LIN {X 0,Y 523.904,Z 120.849,A -85,B 0,C 180,E1 -4806.401,E2 -4806.401} C_VEL
LIN {X 0,Y 523.923,Z 120.845,A -85,B 0,C 180,E1 -4809.085,E2 -4809.085} C_VEL
LIN {X 0,Y 523.952,Z 120.843,A -85,B 0,C 180,E1 -4812.119,E2 -4812.119} C_VEL
LIN {X 0,Y 523.947,Z 120.843,A -85,B 0,C 180,E1 -4815.31,E2 -4815.31} C_VEL
LIN {X 0,Y 523.957,Z 120.839,A -85,B 0,C 180,E1 -4818.69,E2 -4818.69} C_VEL
LIN {X 0,Y 523.918,Z 120.847,A -85,B 0,C 180,E1 -4821.081,E2 -4821.081} C_VEL
LIN {X 0,Y 523.902,Z 120.847,A -85,B 0,C 180,E1 -4823.825,E2 -4823.825} C_VEL
LIN {X 0,Y 523.914,Z 120.844,A -85,B 0,C 180,E1 -4826.634,E2 -4826.634} C_VEL
LIN {X 0,Y 523.95,Z 120.845,A -85,B 0,C 180,E1 -4829.355,E2 -4829.355} C_VEL
LIN {X 0,Y 523.96,Z 120.838,A -85,B 0,C 180,E1 -4832.286,E2 -4832.286} C_VEL
LIN {X 0,Y 523.904,Z 120.849,A -85,B 0,C 180,E1 -4835.427,E2 -4835.427} C_VEL
LIN {X 0,Y 523.94,Z 120.841,A -85,B 0,C 180,E1 -4837.94,E2 -4837.94} C_VEL
LIN {X 0,Y 523.971,Z 120.837,A -85,B 0,C 180,E1 -4840.408,E2 -4840.408} C_VEL
LIN {X 0,Y 523.945,Z 120.848,A -85,B 0,C 180,E1 -4842.837,E2 -4842.837} C_VEL
LIN {X 0,Y 523.976,Z 120.84,A -85,B 0,C 180,E1 -4845.236,E2 -4845.236} C_VEL
LIN {X 0,Y 524.016,Z 120.834,A -85,B 0,C 180,E1 -4848.394,E2 -4848.394} C_VEL
LIN {X 0,Y 523.988,Z 120.833,A -85,B 0,C 180,E1 -4851.516,E2 -4851.516} C_VEL
LIN {X 0,Y 524.069,Z 120.832,A -85,B 0,C 180,E1 -4854.614,E2 -4854.614} C_VEL
LIN {X 0,Y 524.111,Z 120.82,A -85,B 0,C 180,E1 -4857.695,E2 -4857.695} C_VEL
LIN {X 0,Y 524.12,Z 120.822,A -85,B 0,C 180,E1 -4860.768,E2 -4860.768} C_VEL
LIN {X 0,Y 524.006,Z 120.833,A -85,B 0,C 180,E1 -4863.075,E2 -4863.075} C_VEL
LIN {X 0,Y 524.067,Z 120.824,A -85,B 0,C 180,E1 -4865.387,E2 -4865.387} C_VEL
LIN {X 0,Y 523.963,Z 120.84,A -85,B 0,C 180,E1 -4868.485,E2 -4868.485} C_VEL
LIN {X 0,Y 524.001,Z 120.838,A -85,B 0,C 180,E1 -4871.736,E2 -4871.736} C_VEL
LIN {X 0,Y 523.99,Z 120.835,A -85,B 0,C 180,E1 -4875.049,E2 -4875.049} C_VEL
LIN {X 0,Y 523.916,Z 120.852,A -85,B 0,C 180,E1 -4877.971,E2 -4877.971} C_VEL
LIN {X 0,Y 523.951,Z 120.84,A -85,B 0,C 180,E1 -4880.411,E2 -4880.411} C_VEL
LIN {X 0,Y 523.909,Z 120.845,A -85,B 0,C 180,E1 -4882.894,E2 -4882.894} C_VEL
LIN {X 0,Y 523.902,Z 120.849,A -85,B 0,C 180,E1 -4885.421,E2 -4885.421} C_VEL
LIN {X 0,Y 523.907,Z 120.848,A -85,B 0,C 180,E1 -4888.003,E2 -4888.003} C_VEL
LIN {X 0,Y 523.91,Z 120.846,A -85,B 0,C 180,E1 -4890.848,E2 -4890.848} C_VEL
LIN {X 0,Y 523.927,Z 120.846,A -85,B 0,C 180,E1 -4893.729,E2 -4893.729} C_VEL
LIN {X 0,Y 523.888,Z 120.847,A -85,B 0,C 180,E1 -4896.399,E2 -4896.399} C_VEL
LIN {X 0,Y 523.91,Z 120.85,A -85,B 0,C 180,E1 -4899.086,E2 -4899.086} C_VEL
LIN {X 0,Y 523.892,Z 120.846,A -85,B 0,C 180,E1 -4902.125,E2 -4902.125} C_VEL
LIN {X 0,Y 523.935,Z 120.848,A -85,B 0,C 180,E1 -4905.311,E2 -4905.311} C_VEL
LIN {X 0,Y 523.878,Z 120.854,A -85,B 0,C 180,E1 -4906.888,E2 -4906.888} C_VEL
LIN {X 0,Y 523.199,Z 120.937,A -85,B 0,C 180,E1 -4907.529,E2 -4907.529} C_VEL
LIN {X 0,Y 520.357,Z 121.291,A -85,B 0,C 180,E1 -4908.571,E2 -4908.571} C_VEL
LIN {X 0,Y 517.966,Z 121.59,A -85,B 0,C 180,E1 -4909.41,E2 -4909.41} C_VEL
LIN {X 0,Y 516.94,Z 121.715,A -85,B 0,C 180,E1 -4910.058,E2 -4910.058} C_VEL
LIN {X 0,Y 516.856,Z 121.726,A -85,B 0,C 180,E1 -4910.277,E2 -4910.277} C_VEL
LIN {X 0,Y 516.815,Z 121.733,A -85,B 0,C 180,E1 -4913.249,E2 -4913.249} C_VEL
LIN {X 0,Y 516.867,Z 121.725,A -85,B 0,C 180,E1 -4916.117,E2 -4916.117} C_VEL
LIN {X 0,Y 516.848,Z 121.726,A -85,B 0,C 180,E1 -4918.944,E2 -4918.944} C_VEL
LIN {X 0,Y 516.855,Z 121.729,A -85,B 0,C 180,E1 -4922.11,E2 -4922.11} C_VEL
LIN {X 0,Y 516.85,Z 121.746,A -85,B 0,C 180,E1 -4924.907,E2 -4924.907} C_VEL
LIN {X 0,Y 519.11,Z 132.074,A -85,B 0,C 180,E1 -4926.671,E2 -4926.671} C_VEL
LIN {X 0,Y 518.957,Z 140.283,A -85,B 0,C 180,E1 -4927.947,E2 -4927.947} C_VEL
LIN {X 0,Y 518.924,Z 142.324,A -85,B 0,C 180,E1 -4928.26,E2 -4928.26} C_VEL
LIN {X 0,Y 522.001,Z 156.207,A -85,B 0,C 180,E1 -4928.604,E2 -4928.604} C_VEL
LIN {X 0,Y 520.908,Z 307.341,A -85,B 0,C 180,E1 -4930.757,E2 -4930.757} C_VEL
LIN {X 0,Y 520.622,Z 323.147,A -85,B 0,C 180,E1 -4931.147,E2 -4931.147} C_VEL
LIN {X 0,Y 520.269,Z 338.38,A -85,B 0,C 180,E1 -4931.695,E2 -4931.695} C_VEL
LIN {X 0,Y 519.864,Z 351.067,A -85,B 0,C 180,E1 -4932.291,E2 -4932.291} C_VEL
LIN {X 0,Y 519.302,Z 364.673,A -85,B 0,C 180,E1 -4933.084,E2 -4933.084} C_VEL
LIN {X 0,Y 518.776,Z 377.627,A -85,B 0,C 180,E1 -4934.012,E2 -4934.012} C_VEL
LIN {X 0,Y 518.258,Z 389.833,A -85,B 0,C 180,E1 -4935.069,E2 -4935.069} C_VEL
LIN {X 0,Y 517.798,Z 401.302,A -85,B 0,C 180,E1 -4936.259,E2 -4936.259} C_VEL
LIN {X 0,Y 517.363,Z 410.954,A -85,B 0,C 180,E1 -4937.447,E2 -4937.447} C_VEL
LIN {X 0,Y 517.036,Z 420.409,A -85,B 0,C 180,E1 -4938.831,E2 -4938.831} C_VEL
LIN {X 0,Y 516.755,Z 428.281,A -85,B 0,C 180,E1 -4940.212,E2 -4940.212} C_VEL
LIN {X 0,Y 516.546,Z 435.629,A -85,B 0,C 180,E1 -4941.787,E2 -4941.787} C_VEL
LIN {X 0,Y 516.391,Z 441.827,A -85,B 0,C 180,E1 -4943.474,E2 -4943.474} C_VEL
LIN {X 0,Y 516.383,Z 444.913,A -85,B 0,C 180,E1 -4944.533,E2 -4944.533} C_VEL
LIN {X 0,Y 516.327,Z 448.416,A -85,B 0,C 180,E1 -4946.098,E2 -4946.098} C_VEL
LIN {X 0,Y 516.259,Z 450.736,A -85,B 0,C 180,E1 -4947.659,E2 -4947.659} C_VEL
LIN {X 0,Y 516.157,Z 451.927,A -85,B 0,C 180,E1 -4949.22,E2 -4949.22} C_VEL
LIN {X 0,Y 516.158,Z 451.946,A -85,B 0,C 180,E1 -4950.78,E2 -4950.78} C_VEL
LIN {X 0,Y 516.259,Z 450.832,A -85,B 0,C 180,E1 -4952.341,E2 -4952.341} C_VEL
LIN {X 0,Y 516.327,Z 448.586,A -85,B 0,C 180,E1 -4953.902,E2 -4953.902} C_VEL
LIN {X 0,Y 516.38,Z 445.154,A -85,B 0,C 180,E1 -4955.467,E2 -4955.467} C_VEL
LIN {X 0,Y 516.407,Z 440.456,A -85,B 0,C 180,E1 -4957.036,E2 -4957.036} C_VEL
LIN {X 0,Y 516.586,Z 434.365,A -85,B 0,C 180,E1 -4958.607,E2 -4958.607} C_VEL
LIN {X 0,Y 516.804,Z 426.696,A -85,B 0,C 180,E1 -4960.183,E2 -4960.183} C_VEL
LIN {X 0,Y 517.084,Z 418.515,A -85,B 0,C 180,E1 -4961.565,E2 -4961.565} C_VEL
LIN {X 0,Y 517.468,Z 408.661,A -85,B 0,C 180,E1 -4962.95,E2 -4962.95} C_VEL
LIN {X 0,Y 517.877,Z 398.555,A -85,B 0,C 180,E1 -4964.139,E2 -4964.139} C_VEL
LIN {X 0,Y 518.392,Z 386.643,A -85,B 0,C 180,E1 -4965.318,E2 -4965.318} C_VEL
LIN {X 0,Y 518.979,Z 373.3,A -85,B 0,C 180,E1 -4966.411,E2 -4966.411} C_VEL
LIN {X 0,Y 519.534,Z 359.772,A -85,B 0,C 180,E1 -4967.314,E2 -4967.314} C_VEL
LIN {X 0,Y 520.028,Z 344.864,A -85,B 0,C 180,E1 -4968.11,E2 -4968.11} C_VEL
LIN {X 0,Y 520.469,Z 329.611,A -85,B 0,C 180,E1 -4968.731,E2 -4968.731} C_VEL
LIN {X 0,Y 520.798,Z 314.908,A -85,B 0,C 180,E1 -4969.167,E2 -4969.167} C_VEL
LIN {X 0,Y 521,Z 299.457,A -85,B 0,C 180,E1 -4969.463,E2 -4969.463} C_VEL
LIN {X 0,Y 522.003,Z 157.022,A -85,B 0,C 180,E1 -4971.475,E2 -4971.475} C_VEL
LIN {X 0,Y 520.545,Z 149.408,A -85,B 0,C 180,E1 -4971.649,E2 -4971.649} C_VEL
LIN {X 0,Y 518.91,Z 142.309,A -85,B 0,C 180,E1 -4971.832,E2 -4971.832} C_VEL
LIN {X 0,Y 519.187,Z 132.644,A -85,B 0,C 180,E1 -4973.325,E2 -4973.325} C_VEL
LIN {X 0,Y 516.847,Z 121.733,A -85,B 0,C 180,E1 -4975.2,E2 -4975.2} C_VEL
LIN {X 0,Y 516.829,Z 121.731,A -85,B 0,C 180,E1 -4978.421,E2 -4978.421} C_VEL
LIN {X 0,Y 516.848,Z 121.732,A -85,B 0,C 180,E1 -4981.112,E2 -4981.112} C_VEL
LIN {X 0,Y 516.869,Z 121.724,A -85,B 0,C 180,E1 -4983.959,E2 -4983.959} C_VEL
LIN {X 0,Y 516.8,Z 121.735,A -85,B 0,C 180,E1 -4986.753,E2 -4986.753} C_VEL
LIN {X 0,Y 516.825,Z 121.728,A -85,B 0,C 180,E1 -4989.727,E2 -4989.727} C_VEL
LIN {X 0,Y 516.841,Z 121.732,A -85,B 0,C 180,E1 -4992.836,E2 -4992.836} C_VEL
LIN {X 0,Y 516.897,Z 121.727,A -85,B 0,C 180,E1 -4995.007,E2 -4995.007} C_VEL
LIN {X 0,Y 516.847,Z 121.723,A -85,B 0,C 180,E1 -4998.407,E2 -4998.407} C_VEL
LIN {X 0,Y 516.87,Z 121.721,A -85,B 0,C 180,E1 -5001.283,E2 -5001.283} C_VEL
LIN {X 0,Y 516.852,Z 121.731,A -85,B 0,C 180,E1 -5004.673,E2 -5004.673} C_VEL
LIN {X 0,Y 516.893,Z 121.716,A -85,B 0,C 180,E1 -5007.458,E2 -5007.458} C_VEL
LIN {X 0,Y 516.828,Z 121.733,A -85,B 0,C 180,E1 -5010.69,E2 -5010.69} C_VEL
LIN {X 0,Y 516.839,Z 121.725,A -85,B 0,C 180,E1 -5013.337,E2 -5013.337} C_VEL
LIN {X 0,Y 516.884,Z 121.723,A -85,B 0,C 180,E1 -5015.927,E2 -5015.927} C_VEL
LIN {X 0,Y 516.868,Z 121.728,A -85,B 0,C 180,E1 -5018.461,E2 -5018.461} C_VEL
LIN {X 0,Y 516.882,Z 121.72,A -85,B 0,C 180,E1 -5020.954,E2 -5020.954} C_VEL
LIN {X 0,Y 516.834,Z 121.727,A -85,B 0,C 180,E1 -5023.407,E2 -5023.407} C_VEL
LIN {X 0,Y 516.884,Z 121.725,A -85,B 0,C 180,E1 -5025.833,E2 -5025.833} C_VEL
LIN {X 0,Y 516.951,Z 121.712,A -85,B 0,C 180,E1 -5029.028,E2 -5029.028} C_VEL
LIN {X 0,Y 516.927,Z 121.719,A -85,B 0,C 180,E1 -5032.186,E2 -5032.186} C_VEL
LIN {X 0,Y 516.989,Z 121.706,A -85,B 0,C 180,E1 -5034.539,E2 -5034.539} C_VEL
LIN {X 0,Y 517.077,Z 121.704,A -85,B 0,C 180,E1 -5037.663,E2 -5037.663} C_VEL
LIN {X 0,Y 517.072,Z 121.698,A -85,B 0,C 180,E1 -5040,E2 -5040} C_VEL
LIN {X 0,Y 517.082,Z 121.696,A -85,B 0,C 180,E1 -5042.337,E2 -5042.337} C_VEL
LIN {X 0,Y 517.015,Z 121.709,A -85,B 0,C 180,E1 -5045.46,E2 -5045.46} C_VEL
LIN {X 0,Y 516.956,Z 121.711,A -85,B 0,C 180,E1 -5048.6,E2 -5048.6} C_VEL
LIN {X 0,Y 516.956,Z 121.714,A -85,B 0,C 180,E1 -5051.807,E2 -5051.807} C_VEL
LIN {X 0,Y 516.94,Z 121.72,A -85,B 0,C 180,E1 -5055.143,E2 -5055.143} C_VEL
LIN {X 0,Y 516.915,Z 121.714,A -85,B 0,C 180,E1 -5058.222,E2 -5058.222} C_VEL
LIN {X 0,Y 516.908,Z 121.722,A -85,B 0,C 180,E1 -5060.702,E2 -5060.702} C_VEL
LIN {X 0,Y 516.886,Z 121.721,A -85,B 0,C 180,E1 -5064.073,E2 -5064.073} C_VEL
LIN {X 0,Y 516.897,Z 121.723,A -85,B 0,C 180,E1 -5066.659,E2 -5066.659} C_VEL
LIN {X 0,Y 516.911,Z 121.718,A -85,B 0,C 180,E1 -5069.523,E2 -5069.523} C_VEL
LIN {X 0,Y 516.896,Z 121.726,A -85,B 0,C 180,E1 -5072.543,E2 -5072.543} C_VEL
LIN {X 0,Y 516.867,Z 121.723,A -85,B 0,C 180,E1 -5075.329,E2 -5075.329} C_VEL
LIN {X 0,Y 516.881,Z 121.721,A -85,B 0,C 180,E1 -5077.943,E2 -5077.943} C_VEL
LIN {X 0,Y 516.884,Z 121.726,A -85,B 0,C 180,E1 -5080.742,E2 -5080.742} C_VEL
LIN {X 0,Y 516.884,Z 121.724,A -85,B 0,C 180,E1 -5082.831,E2 -5082.831} C_VEL
LIN {X 0,Y 516.896,Z 121.72,A -85,B 0,C 180,E1 -5085.007,E2 -5085.007} C_VEL
LIN {X 0,Y 516.914,Z 121.721,A -85,B 0,C 180,E1 -5088.399,E2 -5088.399} C_VEL
LIN {X 0,Y 516.883,Z 121.721,A -85,B 0,C 180,E1 -5091.284,E2 -5091.284} C_VEL
LIN {X 0,Y 516.872,Z 121.729,A -85,B 0,C 180,E1 -5094.219,E2 -5094.219} C_VEL
LIN {X 0,Y 516.896,Z 121.721,A -85,B 0,C 180,E1 -5097.053,E2 -5097.053} C_VEL
LIN {X 0,Y 516.893,Z 121.725,A -85,B 0,C 180,E1 -5099.796,E2 -5099.796} C_VEL
LIN {X 0,Y 516.97,Z 121.904,A -85,B 0,C 180,E1 -5101.763,E2 -5101.763} C_VEL
LIN {X 0,Y 519.924,Z 134.919,A -85,B 0,C 180,E1 -5103.724,E2 -5103.724} C_VEL
LIN {X 0,Y 519.285,Z 155.389,A -85,B 0,C 180,E1 -5106.468,E2 -5106.468} C_VEL
LIN {X 0,Y 518.846,Z 168.536,A -85,B 0,C 180,E1 -5108.206,E2 -5108.206} C_VEL
LIN {X 0,Y 521.856,Z 183.857,A -85,B 0,C 180,E1 -5108.559,E2 -5108.559} C_VEL
LIN {X 0,Y 520.934,Z 318.473,A -85,B 0,C 180,E1 -5110.458,E2 -5110.458} C_VEL
LIN {X 0,Y 520.766,Z 339.002,A -85,B 0,C 180,E1 -5110.799,E2 -5110.799} C_VEL
LIN {X 0,Y 520.416,Z 353.58,A -85,B 0,C 180,E1 -5111.19,E2 -5111.19} C_VEL
LIN {X 0,Y 519.992,Z 368.148,A -85,B 0,C 180,E1 -5111.736,E2 -5111.736} C_VEL
LIN {X 0,Y 519.528,Z 381.49,A -85,B 0,C 180,E1 -5112.381,E2 -5112.381} C_VEL
LIN {X 0,Y 519.024,Z 394.711,A -85,B 0,C 180,E1 -5113.176,E2 -5113.176} C_VEL
LIN {X 0,Y 518.531,Z 407.433,A -85,B 0,C 180,E1 -5114.108,E2 -5114.108} C_VEL
LIN {X 0,Y 517.946,Z 420.434,A -85,B 0,C 180,E1 -5115.261,E2 -5115.261} C_VEL
LIN {X 0,Y 517.52,Z 431.632,A -85,B 0,C 180,E1 -5116.452,E2 -5116.452} C_VEL
LIN {X 0,Y 517.1,Z 442.501,A -85,B 0,C 180,E1 -5117.839,E2 -5117.839} C_VEL
LIN {X 0,Y 516.872,Z 451.552,A -85,B 0,C 180,E1 -5119.224,E2 -5119.224} C_VEL
LIN {X 0,Y 516.575,Z 459.057,A -85,B 0,C 180,E1 -5120.604,E2 -5120.604} C_VEL
LIN {X 0,Y 516.435,Z 466.064,A -85,B 0,C 180,E1 -5122.178,E2 -5122.178} C_VEL
LIN {X 0,Y 516.36,Z 471.573,A -85,B 0,C 180,E1 -5123.749,E2 -5123.749} C_VEL
LIN {X 0,Y 516.239,Z 475.735,A -85,B 0,C 180,E1 -5125.315,E2 -5125.315} C_VEL
LIN {X 0,Y 516.27,Z 478.657,A -85,B 0,C 180,E1 -5126.879,E2 -5126.879} C_VEL
LIN {X 0,Y 516.189,Z 480.396,A -85,B 0,C 180,E1 -5128.44,E2 -5128.44} C_VEL
LIN {X 0,Y 516.152,Z 480.992,A -85,B 0,C 180,E1 -5130,E2 -5130} C_VEL
LIN {X 0,Y 516.189,Z 480.394,A -85,B 0,C 180,E1 -5131.56,E2 -5131.56} C_VEL
LIN {X 0,Y 516.27,Z 478.652,A -85,B 0,C 180,E1 -5133.121,E2 -5133.121} C_VEL
LIN {X 0,Y 516.239,Z 475.733,A -85,B 0,C 180,E1 -5134.685,E2 -5134.685} C_VEL
LIN {X 0,Y 516.365,Z 471.577,A -85,B 0,C 180,E1 -5136.251,E2 -5136.251} C_VEL
LIN {X 0,Y 516.435,Z 466.065,A -85,B 0,C 180,E1 -5137.821,E2 -5137.821} C_VEL
LIN {X 0,Y 516.575,Z 459.051,A -85,B 0,C 180,E1 -5139.396,E2 -5139.396} C_VEL
LIN {X 0,Y 516.858,Z 451.548,A -85,B 0,C 180,E1 -5140.776,E2 -5140.776} C_VEL
LIN {X 0,Y 517.089,Z 442.772,A -85,B 0,C 180,E1 -5142.122,E2 -5142.122} C_VEL
LIN {X 0,Y 517.473,Z 433.272,A -85,B 0,C 180,E1 -5143.349,E2 -5143.349} C_VEL
LIN {X 0,Y 517.871,Z 422.4,A -85,B 0,C 180,E1 -5144.54,E2 -5144.54} C_VEL
LIN {X 0,Y 518.336,Z 411.334,A -85,B 0,C 180,E1 -5145.565,E2 -5145.565} C_VEL
LIN {X 0,Y 518.829,Z 399.006,A -85,B 0,C 180,E1 -5146.527,E2 -5146.527} C_VEL
LIN {X 0,Y 519.381,Z 386.798,A -85,B 0,C 180,E1 -5147.319,E2 -5147.319} C_VEL
LIN {X 0,Y 519.837,Z 372.671,A -85,B 0,C 180,E1 -5148.066,E2 -5148.066} C_VEL
LIN {X 0,Y 520.323,Z 358.14,A -85,B 0,C 180,E1 -5148.66,E2 -5148.66} C_VEL
LIN {X 0,Y 520.674,Z 342.45,A -85,B 0,C 180,E1 -5149.127,E2 -5149.127} C_VEL
LIN {X 0,Y 520.934,Z 326.359,A -85,B 0,C 180,E1 -5149.429,E2 -5149.429} C_VEL
LIN {X 0,Y 521.902,Z 184.332,A -85,B 0,C 180,E1 -5151.432,E2 -5151.432} C_VEL
LIN {X 0,Y 518.854,Z 168.468,A -85,B 0,C 180,E1 -5151.798,E2 -5151.798} C_VEL
LIN {X 0,Y 519.503,Z 149.094,A -85,B 0,C 180,E1 -5154.369,E2 -5154.369} C_VEL
LIN {X 0,Y 519.914,Z 134.915,A -85,B 0,C 180,E1 -5156.276,E2 -5156.276} C_VEL
LIN {X 0,Y 516.925,Z 121.723,A -85,B 0,C 180,E1 -5158.275,E2 -5158.275} C_VEL
LIN {X 0,Y 516.89,Z 121.721,A -85,B 0,C 180,E1 -5161.11,E2 -5161.11} C_VEL
LIN {X 0,Y 516.908,Z 121.723,A -85,B 0,C 180,E1 -5163.966,E2 -5163.966} C_VEL
LIN {X 0,Y 516.877,Z 121.722,A -85,B 0,C 180,E1 -5166.746,E2 -5166.746} C_VEL
LIN {X 0,Y 516.883,Z 121.727,A -85,B 0,C 180,E1 -5169.721,E2 -5169.721} C_VEL
LIN {X 0,Y 516.912,Z 121.725,A -85,B 0,C 180,E1 -5171.775,E2 -5171.775} C_VEL
LIN {X 0,Y 516.896,Z 121.719,A -85,B 0,C 180,E1 -5175.007,E2 -5175.007} C_VEL
LIN {X 0,Y 516.914,Z 121.716,A -85,B 0,C 180,E1 -5178.399,E2 -5178.399} C_VEL
LIN {X 0,Y 516.881,Z 121.726,A -85,B 0,C 180,E1 -5181.284,E2 -5181.284} C_VEL
LIN {X 0,Y 516.872,Z 121.72,A -85,B 0,C 180,E1 -5184.22,E2 -5184.22} C_VEL
LIN {X 0,Y 516.882,Z 121.724,A -85,B 0,C 180,E1 -5187.052,E2 -5187.052} C_VEL
LIN {X 0,Y 516.888,Z 121.72,A -85,B 0,C 180,E1 -5189.796,E2 -5189.796} C_VEL
LIN {X 0,Y 516.912,Z 121.717,A -85,B 0,C 180,E1 -5192.467,E2 -5192.467} C_VEL
LIN {X 0,Y 516.874,Z 121.722,A -85,B 0,C 180,E1 -5195.645,E2 -5195.645} C_VEL
LIN {X 0,Y 516.887,Z 121.722,A -85,B 0,C 180,E1 -5198.462,E2 -5198.462} C_VEL
LIN {X 0,Y 516.894,Z 121.726,A -85,B 0,C 180,E1 -5200.955,E2 -5200.955} C_VEL
LIN {X 0,Y 516.899,Z 121.718,A -85,B 0,C 180,E1 -5203.41,E2 -5203.41} C_VEL
LIN {X 0,Y 516.885,Z 121.72,A -85,B 0,C 180,E1 -5205.833,E2 -5205.833} C_VEL
LIN {X 0,Y 516.952,Z 121.716,A -85,B 0,C 180,E1 -5209.028,E2 -5209.028} C_VEL
LIN {X 0,Y 516.946,Z 121.713,A -85,B 0,C 180,E1 -5212.186,E2 -5212.186} C_VEL
LIN {X 0,Y 517.015,Z 121.711,A -85,B 0,C 180,E1 -5214.54,E2 -5214.54} C_VEL
LIN {X 0,Y 517.082,Z 121.696,A -85,B 0,C 180,E1 -5217.663,E2 -5217.663} C_VEL
LIN {X 0,Y 517.091,Z 121.697,A -85,B 0,C 180,E1 -5220.779,E2 -5220.779} C_VEL
LIN {X 0,Y 516.95,Z 121.712,A -85,B 0,C 180,E1 -5223.117,E2 -5223.117} C_VEL
LIN {X 0,Y 516.974,Z 121.717,A -85,B 0,C 180,E1 -5226.244,E2 -5226.244} C_VEL
LIN {X 0,Y 516.939,Z 121.711,A -85,B 0,C 180,E1 -5229.39,E2 -5229.39} C_VEL
LIN {X 0,Y 516.955,Z 121.717,A -85,B 0,C 180,E1 -5231.807,E2 -5231.807} C_VEL
LIN {X 0,Y 516.942,Z 121.713,A -85,B 0,C 180,E1 -5235.144,E2 -5235.144} C_VEL
LIN {X 0,Y 516.878,Z 121.725,A -85,B 0,C 180,E1 -5238.224,E2 -5238.224} C_VEL
LIN {X 0,Y 516.9,Z 121.717,A -85,B 0,C 180,E1 -5240.702,E2 -5240.702} C_VEL
LIN {X 0,Y 516.858,Z 121.726,A -85,B 0,C 180,E1 -5243.224,E2 -5243.224} C_VEL
LIN {X 0,Y 516.883,Z 121.714,A -85,B 0,C 180,E1 -5246.182,E2 -5246.182} C_VEL
LIN {X 0,Y 516.905,Z 121.722,A -85,B 0,C 180,E1 -5249.306,E2 -5249.306} C_VEL
LIN {X 0,Y 516.893,Z 121.719,A -85,B 0,C 180,E1 -5252.542,E2 -5252.542} C_VEL
LIN {X 0,Y 516.856,Z 121.73,A -85,B 0,C 180,E1 -5255.328,E2 -5255.328} C_VEL
LIN {X 0,Y 516.877,Z 121.722,A -85,B 0,C 180,E1 -5257.942,E2 -5257.942} C_VEL
LIN {X 0,Y 516.848,Z 121.726,A -85,B 0,C 180,E1 -5260.745,E2 -5260.745} C_VEL
LIN {X 0,Y 516.881,Z 121.721,A -85,B 0,C 180,E1 -5263.903,E2 -5263.903} C_VEL
LIN {X 0,Y 516.835,Z 121.73,A -85,B 0,C 180,E1 -5266.888,E2 -5266.888} C_VEL
LIN {X 0,Y 516.859,Z 121.726,A -85,B 0,C 180,E1 -5269.593,E2 -5269.593} C_VEL
LIN {X 0,Y 516.856,Z 121.726,A -85,B 0,C 180,E1 -5270.277,E2 -5270.277} C_VEL
LIN {X 0,Y 516.186,Z 121.812,A -85,B 0,C 180,E1 -5270.927,E2 -5270.927} C_VEL
LIN {X 0,Y 513.32,Z 122.169,A -85,B 0,C 180,E1 -5271.982,E2 -5271.982} C_VEL
LIN {X 0,Y 510.897,Z 122.474,A -85,B 0,C 180,E1 -5272.832,E2 -5272.832} C_VEL
LIN {X 0,Y 509.855,Z 122.598,A -85,B 0,C 180,E1 -5273.489,E2 -5273.489} C_VEL
LIN {X 0,Y 509.769,Z 122.607,A -85,B 0,C 180,E1 -5273.711,E2 -5273.711} C_VEL
LIN {X 0,Y 509.824,Z 122.606,A -85,B 0,C 180,E1 -5276.536,E2 -5276.536} C_VEL
LIN {X 0,Y 509.801,Z 122.599,A -85,B 0,C 180,E1 -5279.331,E2 -5279.331} C_VEL
LIN {X 0,Y 509.822,Z 122.605,A -85,B 0,C 180,E1 -5282.05,E2 -5282.05} C_VEL
LIN {X 0,Y 509.826,Z 122.769,A -85,B 0,C 180,E1 -5284.674,E2 -5284.674} C_VEL
LIN {X 0,Y 512.223,Z 133.604,A -85,B 0,C 180,E1 -5286.553,E2 -5286.553} C_VEL
LIN {X 0,Y 512.211,Z 138.98,A -85,B 0,C 180,E1 -5287.407,E2 -5287.407} C_VEL
LIN {X 0,Y 512.063,Z 142.508,A -85,B 0,C 180,E1 -5287.951,E2 -5287.951} C_VEL
LIN {X 0,Y 515.364,Z 156.872,A -85,B 0,C 180,E1 -5288.32,E2 -5288.32} C_VEL
LIN {X 0,Y 514.4,Z 284.989,A -85,B 0,C 180,E1 -5290.154,E2 -5290.154} C_VEL
LIN {X 0,Y 514.17,Z 309.47,A -85,B 0,C 180,E1 -5290.538,E2 -5290.538} C_VEL
LIN {X 0,Y 513.881,Z 324.887,A -85,B 0,C 180,E1 -5290.942,E2 -5290.942} C_VEL
LIN {X 0,Y 513.499,Z 339.718,A -85,B 0,C 180,E1 -5291.497,E2 -5291.497} C_VEL
LIN {X 0,Y 513.045,Z 353.179,A -85,B 0,C 180,E1 -5292.151,E2 -5292.151} C_VEL
LIN {X 0,Y 512.46,Z 366.447,A -85,B 0,C 180,E1 -5292.954,E2 -5292.954} C_VEL
LIN {X 0,Y 511.837,Z 380.179,A -85,B 0,C 180,E1 -5293.98,E2 -5293.98} C_VEL
LIN {X 0,Y 511.288,Z 392.149,A -85,B 0,C 180,E1 -5295.064,E2 -5295.064} C_VEL
LIN {X 0,Y 510.805,Z 403.276,A -85,B 0,C 180,E1 -5296.271,E2 -5296.271} C_VEL
LIN {X 0,Y 510.278,Z 414.357,A -85,B 0,C 180,E1 -5297.714,E2 -5297.714} C_VEL
LIN {X 0,Y 509.98,Z 423.052,A -85,B 0,C 180,E1 -5299.077,E2 -5299.077} C_VEL
LIN {X 0,Y 509.678,Z 430.483,A -85,B 0,C 180,E1 -5300.475,E2 -5300.475} C_VEL
LIN {X 0,Y 509.453,Z 437.431,A -85,B 0,C 180,E1 -5302.071,E2 -5302.071} C_VEL
LIN {X 0,Y 509.315,Z 442.893,A -85,B 0,C 180,E1 -5303.662,E2 -5303.662} C_VEL
LIN {X 0,Y 509.166,Z 447.02,A -85,B 0,C 180,E1 -5305.249,E2 -5305.249} C_VEL
LIN {X 0,Y 509.189,Z 449.92,A -85,B 0,C 180,E1 -5306.835,E2 -5306.835} C_VEL
LIN {X 0,Y 509.11,Z 451.67,A -85,B 0,C 180,E1 -5308.418,E2 -5308.418} C_VEL
LIN {X 0,Y 509.066,Z 452.284,A -85,B 0,C 180,E1 -5310,E2 -5310} C_VEL
LIN {X 0,Y 509.111,Z 451.727,A -85,B 0,C 180,E1 -5311.582,E2 -5311.582} C_VEL
LIN {X 0,Y 509.19,Z 450.051,A -85,B 0,C 180,E1 -5313.165,E2 -5313.165} C_VEL
LIN {X 0,Y 509.165,Z 447.223,A -85,B 0,C 180,E1 -5314.751,E2 -5314.751} C_VEL
LIN {X 0,Y 509.307,Z 443.168,A -85,B 0,C 180,E1 -5316.338,E2 -5316.338} C_VEL
LIN {X 0,Y 509.453,Z 437.791,A -85,B 0,C 180,E1 -5317.929,E2 -5317.929} C_VEL
LIN {X 0,Y 509.666,Z 430.939,A -85,B 0,C 180,E1 -5319.525,E2 -5319.525} C_VEL
LIN {X 0,Y 509.965,Z 422.384,A -85,B 0,C 180,E1 -5321.124,E2 -5321.124} C_VEL
LIN {X 0,Y 510.326,Z 413.291,A -85,B 0,C 180,E1 -5322.527,E2 -5322.527} C_VEL
LIN {X 0,Y 510.749,Z 404.014,A -85,B 0,C 180,E1 -5323.731,E2 -5323.731} C_VEL
LIN {X 0,Y 511.279,Z 392.026,A -85,B 0,C 180,E1 -5325.038,E2 -5325.038} C_VEL
LIN {X 0,Y 511.915,Z 379.005,A -85,B 0,C 180,E1 -5326.204,E2 -5326.204} C_VEL
LIN {X 0,Y 512.476,Z 366.26,A -85,B 0,C 180,E1 -5327.148,E2 -5327.148} C_VEL
LIN {X 0,Y 513.014,Z 352.963,A -85,B 0,C 180,E1 -5327.953,E2 -5327.953} C_VEL
LIN {X 0,Y 513.555,Z 338.286,A -85,B 0,C 180,E1 -5328.656,E2 -5328.656} C_VEL
LIN {X 0,Y 513.941,Z 323.44,A -85,B 0,C 180,E1 -5329.194,E2 -5329.194} C_VEL
LIN {X 0,Y 514.232,Z 307.532,A -85,B 0,C 180,E1 -5329.593,E2 -5329.593} C_VEL
LIN {X 0,Y 515.379,Z 157.183,A -85,B 0,C 180,E1 -5331.765,E2 -5331.765} C_VEL
LIN {X 0,Y 512.066,Z 142.467,A -85,B 0,C 180,E1 -5332.144,E2 -5332.144} C_VEL
LIN {X 0,Y 512.317,Z 134.163,A -85,B 0,C 180,E1 -5333.442,E2 -5333.442} C_VEL
LIN {X 0,Y 509.801,Z 122.612,A -85,B 0,C 180,E1 -5335.464,E2 -5335.464} C_VEL
LIN {X 0,Y 509.808,Z 122.607,A -85,B 0,C 180,E1 -5338.082,E2 -5338.082} C_VEL
LIN {X 0,Y 509.815,Z 122.609,A -85,B 0,C 180,E1 -5341.274,E2 -5341.274} C_VEL
LIN {X 0,Y 509.821,Z 122.602,A -85,B 0,C 180,E1 -5344.416,E2 -5344.416} C_VEL
LIN {X 0,Y 509.763,Z 122.616,A -85,B 0,C 180,E1 -5347.346,E2 -5347.346} C_VEL
LIN {X 0,Y 509.787,Z 122.604,A -85,B 0,C 180,E1 -5350.387,E2 -5350.387} C_VEL
LIN {X 0,Y 509.793,Z 122.606,A -85,B 0,C 180,E1 -5353.575,E2 -5353.575} C_VEL
LIN {X 0,Y 509.792,Z 122.607,A -85,B 0,C 180,E1 -5356.425,E2 -5356.425} C_VEL
LIN {X 0,Y 509.813,Z 122.602,A -85,B 0,C 180,E1 -5359.615,E2 -5359.615} C_VEL
LIN {X 0,Y 509.784,Z 122.605,A -85,B 0,C 180,E1 -5362.656,E2 -5362.656} C_VEL
LIN {X 0,Y 509.84,Z 122.598,A -85,B 0,C 180,E1 -5365.801,E2 -5365.801} C_VEL
LIN {X 0,Y 509.818,Z 122.598,A -85,B 0,C 180,E1 -5368.726,E2 -5368.726} C_VEL
LIN {X 0,Y 509.824,Z 122.603,A -85,B 0,C 180,E1 -5372.05,E2 -5372.05} C_VEL
LIN {X 0,Y 509.803,Z 122.607,A -85,B 0,C 180,E1 -5374.7,E2 -5374.7} C_VEL
LIN {X 0,Y 509.826,Z 122.598,A -85,B 0,C 180,E1 -5377.459,E2 -5377.459} C_VEL
LIN {X 0,Y 509.892,Z 122.595,A -85,B 0,C 180,E1 -5379.844,E2 -5379.844} C_VEL
LIN {X 0,Y 509.849,Z 122.602,A -85,B 0,C 180,E1 -5382.346,E2 -5382.346} C_VEL
LIN {X 0,Y 509.893,Z 122.591,A -85,B 0,C 180,E1 -5384.818,E2 -5384.818} C_VEL
LIN {X 0,Y 509.905,Z 122.597,A -85,B 0,C 180,E1 -5388.124,E2 -5388.124} C_VEL
LIN {X 0,Y 509.887,Z 122.59,A -85,B 0,C 180,E1 -5391.279,E2 -5391.279} C_VEL
LIN {X 0,Y 509.944,Z 122.584,A -85,B 0,C 180,E1 -5394.464,E2 -5394.464} C_VEL
LIN {X 0,Y 510.046,Z 122.579,A -85,B 0,C 180,E1 -5397.631,E2 -5397.631} C_VEL
LIN {X 0,Y 510.041,Z 122.574,A -85,B 0,C 180,E1 -5400,E2 -5400} C_VEL
LIN {X 0,Y 510.052,Z 122.572,A -85,B 0,C 180,E1 -5402.369,E2 -5402.369} C_VEL
LIN {X 0,Y 509.966,Z 122.588,A -85,B 0,C 180,E1 -5405.536,E2 -5405.536} C_VEL
LIN {X 0,Y 509.905,Z 122.59,A -85,B 0,C 180,E1 -5408.72,E2 -5408.72} C_VEL
LIN {X 0,Y 509.907,Z 122.591,A -85,B 0,C 180,E1 -5411.931,E2 -5411.931} C_VEL
LIN {X 0,Y 509.898,Z 122.599,A -85,B 0,C 180,E1 -5415.242,E2 -5415.242} C_VEL
LIN {X 0,Y 509.86,Z 122.594,A -85,B 0,C 180,E1 -5418.484,E2 -5418.484} C_VEL
LIN {X 0,Y 509.849,Z 122.605,A -85,B 0,C 180,E1 -5421.002,E2 -5421.002} C_VEL
LIN {X 0,Y 509.82,Z 122.602,A -85,B 0,C 180,E1 -5423.564,E2 -5423.564} C_VEL
LIN {X 0,Y 509.876,Z 122.594,A -85,B 0,C 180,E1 -5426.369,E2 -5426.369} C_VEL
LIN {X 0,Y 509.854,Z 122.604,A -85,B 0,C 180,E1 -5428.846,E2 -5428.846} C_VEL
LIN {X 0,Y 509.821,Z 122.601,A -85,B 0,C 180,E1 -5431.59,E2 -5431.59} C_VEL
LIN {X 0,Y 509.84,Z 122.6,A -85,B 0,C 180,E1 -5434.414,E2 -5434.414} C_VEL
LIN {X 0,Y 509.818,Z 122.6,A -85,B 0,C 180,E1 -5437.341,E2 -5437.341} C_VEL
LIN {X 0,Y 509.84,Z 122.603,A -85,B 0,C 180,E1 -5440.382,E2 -5440.382} C_VEL
LIN {X 0,Y 509.824,Z 122.601,A -85,B 0,C 180,E1 -5443.062,E2 -5443.062} C_VEL
LIN {X 0,Y 509.824,Z 122.602,A -85,B 0,C 180,E1 -5445.793,E2 -5445.793} C_VEL
LIN {X 0,Y 509.856,Z 122.597,A -85,B 0,C 180,E1 -5448.574,E2 -5448.574} C_VEL
LIN {X 0,Y 509.852,Z 122.6,A -85,B 0,C 180,E1 -5451.786,E2 -5451.786} C_VEL
LIN {X 0,Y 509.831,Z 122.602,A -85,B 0,C 180,E1 -5454.622,E2 -5454.622} C_VEL
LIN {X 0,Y 509.862,Z 122.599,A -85,B 0,C 180,E1 -5457.481,E2 -5457.481} C_VEL
LIN {X 0,Y 509.86,Z 122.602,A -85,B 0,C 180,E1 -5460.274,E2 -5460.274} C_VEL
LIN {X 0,Y 509.89,Z 122.695,A -85,B 0,C 180,E1 -5461.474,E2 -5461.474} C_VEL
LIN {X 0,Y 513.048,Z 136.31,A -85,B 0,C 180,E1 -5463.564,E2 -5463.564} C_VEL
LIN {X 0,Y 512.528,Z 153.629,A -85,B 0,C 180,E1 -5465.924,E2 -5465.924} C_VEL
LIN {X 0,Y 512.008,Z 168.292,A -85,B 0,C 180,E1 -5467.897,E2 -5467.897} C_VEL
LIN {X 0,Y 515.283,Z 185.415,A -85,B 0,C 180,E1 -5468.297,E2 -5468.297} C_VEL
LIN {X 0,Y 514.141,Z 334.566,A -85,B 0,C 180,E1 -5470.446,E2 -5470.446} C_VEL
LIN {X 0,Y 513.801,Z 350.317,A -85,B 0,C 180,E1 -5470.835,E2 -5470.835} C_VEL
LIN {X 0,Y 513.386,Z 364.448,A -85,B 0,C 180,E1 -5471.337,E2 -5471.337} C_VEL
LIN {X 0,Y 512.782,Z 379.472,A -85,B 0,C 180,E1 -5472.038,E2 -5472.038} C_VEL
LIN {X 0,Y 512.234,Z 392.989,A -85,B 0,C 180,E1 -5472.843,E2 -5472.843} C_VEL
LIN {X 0,Y 511.707,Z 405.456,A -85,B 0,C 180,E1 -5473.749,E2 -5473.749} C_VEL
LIN {X 0,Y 511.153,Z 418.137,A -85,B 0,C 180,E1 -5474.856,E2 -5474.856} C_VEL
LIN {X 0,Y 510.615,Z 429.658,A -85,B 0,C 180,E1 -5476.062,E2 -5476.062} C_VEL
LIN {X 0,Y 510.205,Z 439.359,A -85,B 0,C 180,E1 -5477.268,E2 -5477.268} C_VEL
LIN {X 0,Y 509.83,Z 449.043,A -85,B 0,C 180,E1 -5478.697,E2 -5478.697} C_VEL
LIN {X 0,Y 509.562,Z 456.826,A -85,B 0,C 180,E1 -5480.072,E2 -5480.072} C_VEL
LIN {X 0,Y 509.394,Z 464.24,A -85,B 0,C 180,E1 -5481.67,E2 -5481.67} C_VEL
LIN {X 0,Y 509.289,Z 470.122,A -85,B 0,C 180,E1 -5483.264,E2 -5483.264} C_VEL
LIN {X 0,Y 509.263,Z 473.617,A -85,B 0,C 180,E1 -5484.456,E2 -5484.456} C_VEL
LIN {X 0,Y 509.172,Z 477.148,A -85,B 0,C 180,E1 -5486.043,E2 -5486.043} C_VEL
LIN {X 0,Y 509.186,Z 479.473,A -85,B 0,C 180,E1 -5487.627,E2 -5487.627} C_VEL
LIN {X 0,Y 509.07,Z 480.64,A -85,B 0,C 180,E1 -5489.209,E2 -5489.209} C_VEL
LIN {X 0,Y 509.07,Z 480.639,A -85,B 0,C 180,E1 -5490.791,E2 -5490.791} C_VEL
LIN {X 0,Y 509.186,Z 479.469,A -85,B 0,C 180,E1 -5492.373,E2 -5492.373} C_VEL
LIN {X 0,Y 509.172,Z 477.144,A -85,B 0,C 180,E1 -5493.957,E2 -5493.957} C_VEL
LIN {X 0,Y 509.264,Z 473.618,A -85,B 0,C 180,E1 -5495.544,E2 -5495.544} C_VEL
LIN {X 0,Y 509.315,Z 468.799,A -85,B 0,C 180,E1 -5497.134,E2 -5497.134} C_VEL
LIN {X 0,Y 509.453,Z 462.557,A -85,B 0,C 180,E1 -5498.728,E2 -5498.728} C_VEL
LIN {X 0,Y 509.701,Z 454.72,A -85,B 0,C 180,E1 -5500.326,E2 -5500.326} C_VEL
LIN {X 0,Y 509.937,Z 446.321,A -85,B 0,C 180,E1 -5501.738,E2 -5501.738} C_VEL
LIN {X 0,Y 510.339,Z 436.344,A -85,B 0,C 180,E1 -5503.134,E2 -5503.134} C_VEL
LIN {X 0,Y 510.755,Z 426.075,A -85,B 0,C 180,E1 -5504.34,E2 -5504.34} C_VEL
LIN {X 0,Y 511.33,Z 413.429,A -85,B 0,C 180,E1 -5505.585,E2 -5505.585} C_VEL
LIN {X 0,Y 511.917,Z 400.238,A -85,B 0,C 180,E1 -5506.654,E2 -5506.654} C_VEL
LIN {X 0,Y 512.577,Z 386.598,A -85,B 0,C 180,E1 -5507.556,E2 -5507.556} C_VEL
LIN {X 0,Y 513.067,Z 372.471,A -85,B 0,C 180,E1 -5508.312,E2 -5508.312} C_VEL
LIN {X 0,Y 513.586,Z 357.969,A -85,B 0,C 180,E1 -5508.913,E2 -5508.913} C_VEL
LIN {X 0,Y 513.951,Z 342.522,A -85,B 0,C 180,E1 -5509.381,E2 -5509.381} C_VEL
LIN {X 0,Y 514.239,Z 326.159,A -85,B 0,C 180,E1 -5509.693,E2 -5509.693} C_VEL
LIN {X 0,Y 515.303,Z 185.412,A -85,B 0,C 180,E1 -5511.702,E2 -5511.702} C_VEL
LIN {X 0,Y 511.998,Z 168.264,A -85,B 0,C 180,E1 -5512.106,E2 -5512.106} C_VEL
LIN {X 0,Y 512.71,Z 148.903,A -85,B 0,C 180,E1 -5514.714,E2 -5514.714} C_VEL
LIN {X 0,Y 513.037,Z 136.304,A -85,B 0,C 180,E1 -5516.437,E2 -5516.437} C_VEL
LIN {X 0,Y 509.895,Z 122.599,A -85,B 0,C 180,E1 -5518.55,E2 -5518.55} C_VEL
LIN {X 0,Y 509.821,Z 122.603,A -85,B 0,C 180,E1 -5521.59,E2 -5521.59} C_VEL
LIN {X 0,Y 509.848,Z 122.6,A -85,B 0,C 180,E1 -5524.414,E2 -5524.414} C_VEL
LIN {X 0,Y 509.818,Z 122.603,A -85,B 0,C 180,E1 -5527.341,E2 -5527.341} C_VEL
LIN {X 0,Y 509.839,Z 122.6,A -85,B 0,C 180,E1 -5530.382,E2 -5530.382} C_VEL
LIN {X 0,Y 509.825,Z 122.6,A -85,B 0,C 180,E1 -5533.062,E2 -5533.062} C_VEL
LIN {X 0,Y 509.824,Z 122.606,A -85,B 0,C 180,E1 -5535.793,E2 -5535.793} C_VEL
LIN {X 0,Y 509.856,Z 122.595,A -85,B 0,C 180,E1 -5538.575,E2 -5538.575} C_VEL
LIN {X 0,Y 509.852,Z 122.6,A -85,B 0,C 180,E1 -5541.787,E2 -5541.787} C_VEL
LIN {X 0,Y 509.83,Z 122.597,A -85,B 0,C 180,E1 -5544.622,E2 -5544.622} C_VEL
LIN {X 0,Y 509.861,Z 122.601,A -85,B 0,C 180,E1 -5547.481,E2 -5547.481} C_VEL
LIN {X 0,Y 509.86,Z 122.593,A -85,B 0,C 180,E1 -5550.274,E2 -5550.274} C_VEL
LIN {X 0,Y 509.868,Z 122.599,A -85,B 0,C 180,E1 -5552.943,E2 -5552.943} C_VEL
LIN {X 0,Y 509.82,Z 122.6,A -85,B 0,C 180,E1 -5556.436,E2 -5556.436} C_VEL
LIN {X 0,Y 509.917,Z 122.586,A -85,B 0,C 180,E1 -5559.845,E2 -5559.845} C_VEL
LIN {X 0,Y 509.866,Z 122.597,A -85,B 0,C 180,E1 -5563.174,E2 -5563.174} C_VEL
LIN {X 0,Y 509.857,Z 122.596,A -85,B 0,C 180,E1 -5565.634,E2 -5565.634} C_VEL
LIN {X 0,Y 509.915,Z 122.595,A -85,B 0,C 180,E1 -5568.875,E2 -5568.875} C_VEL
LIN {X 0,Y 509.911,Z 122.588,A -85,B 0,C 180,E1 -5572.078,E2 -5572.078} C_VEL
LIN {X 0,Y 509.966,Z 122.59,A -85,B 0,C 180,E1 -5574.464,E2 -5574.464} C_VEL
LIN {X 0,Y 510.052,Z 122.571,A -85,B 0,C 180,E1 -5577.631,E2 -5577.631} C_VEL
LIN {X 0,Y 510.041,Z 122.575,A -85,B 0,C 180,E1 -5580.79,E2 -5580.79} C_VEL
LIN {X 0,Y 510.047,Z 122.58,A -85,B 0,C 180,E1 -5582.369,E2 -5582.369} C_VEL
LIN {X 0,Y 509.964,Z 122.581,A -85,B 0,C 180,E1 -5585.536,E2 -5585.536} C_VEL
LIN {X 0,Y 509.891,Z 122.59,A -85,B 0,C 180,E1 -5588.721,E2 -5588.721} C_VEL
LIN {X 0,Y 509.907,Z 122.596,A -85,B 0,C 180,E1 -5591.932,E2 -5591.932} C_VEL
LIN {X 0,Y 509.898,Z 122.591,A -85,B 0,C 180,E1 -5595.242,E2 -5595.242} C_VEL
LIN {X 0,Y 509.836,Z 122.6,A -85,B 0,C 180,E1 -5598.485,E2 -5598.485} C_VEL
LIN {X 0,Y 509.843,Z 122.596,A -85,B 0,C 180,E1 -5601.002,E2 -5601.002} C_VEL
LIN {X 0,Y 509.82,Z 122.607,A -85,B 0,C 180,E1 -5603.564,E2 -5603.564} C_VEL
LIN {X 0,Y 509.819,Z 122.592,A -85,B 0,C 180,E1 -5606.357,E2 -5606.357} C_VEL
LIN {X 0,Y 509.838,Z 122.598,A -85,B 0,C 180,E1 -5608.847,E2 -5608.847} C_VEL
LIN {X 0,Y 509.814,Z 122.607,A -85,B 0,C 180,E1 -5611.591,E2 -5611.591} C_VEL
LIN {X 0,Y 509.835,Z 122.596,A -85,B 0,C 180,E1 -5614.415,E2 -5614.415} C_VEL
LIN {X 0,Y 509.807,Z 122.608,A -85,B 0,C 180,E1 -5617.342,E2 -5617.342} C_VEL
LIN {X 0,Y 509.813,Z 122.6,A -85,B 0,C 180,E1 -5620.385,E2 -5620.385} C_VEL
LIN {X 0,Y 509.806,Z 122.605,A -85,B 0,C 180,E1 -5623.573,E2 -5623.573} C_VEL
LIN {X 0,Y 509.806,Z 122.603,A -85,B 0,C 180,E1 -5626.426,E2 -5626.426} C_VEL
LIN {X 0,Y 509.813,Z 122.604,A -85,B 0,C 180,E1 -5629.615,E2 -5629.615} C_VEL
LIN {X 0,Y 509.783,Z 122.61,A -85,B 0,C 180,E1 -5632.656,E2 -5632.656} C_VEL
LIN {X 0,Y 509.769,Z 122.607,A -85,B 0,C 180,E1 -5633.711,E2 -5633.711} C_VEL
LIN {X 0,Y 509.109,Z 122.692,A -85,B 0,C 180,E1 -5634.371,E2 -5634.371} C_VEL
LIN {X 0,Y 506.284,Z 123.045,A -85,B 0,C 180,E1 -5635.444,E2 -5635.444} C_VEL
LIN {X 0,Y 503.888,Z 123.345,A -85,B 0,C 180,E1 -5636.307,E2 -5636.307} C_VEL
LIN {X 0,Y 502.847,Z 123.473,A -85,B 0,C 180,E1 -5636.974,E2 -5636.974} C_VEL
LIN {X 0,Y 502.756,Z 123.483,A -85,B 0,C 180,E1 -5637.2,E2 -5637.2} C_VEL
LIN {X 0,Y 502.744,Z 123.476,A -85,B 0,C 180,E1 -5640.079,E2 -5640.079} C_VEL
LIN {X 0,Y 502.768,Z 123.485,A -85,B 0,C 180,E1 -5642.529,E2 -5642.529} C_VEL
LIN {X 0,Y 502.783,Z 123.616,A -85,B 0,C 180,E1 -5644.404,E2 -5644.404} C_VEL
LIN {X 0,Y 505.474,Z 136.043,A -85,B 0,C 180,E1 -5646.585,E2 -5646.585} C_VEL
LIN {X 0,Y 505.253,Z 142.701,A -85,B 0,C 180,E1 -5647.638,E2 -5647.638} C_VEL
LIN {X 0,Y 508.834,Z 158.982,A -85,B 0,C 180,E1 -5648.056,E2 -5648.056} C_VEL
LIN {X 0,Y 507.56,Z 308.005,A -85,B 0,C 180,E1 -5650.235,E2 -5650.235} C_VEL
LIN {X 0,Y 507.218,Z 323.58,A -85,B 0,C 180,E1 -5650.629,E2 -5650.629} C_VEL
LIN {X 0,Y 506.82,Z 338.804,A -85,B 0,C 180,E1 -5651.192,E2 -5651.192} C_VEL
LIN {X 0,Y 506.353,Z 351.488,A -85,B 0,C 180,E1 -5651.803,E2 -5651.803} C_VEL
LIN {X 0,Y 505.72,Z 365.091,A -85,B 0,C 180,E1 -5652.615,E2 -5652.615} C_VEL
LIN {X 0,Y 505.142,Z 377.723,A -85,B 0,C 180,E1 -5653.543,E2 -5653.543} C_VEL
LIN {X 0,Y 504.484,Z 390.246,A -85,B 0,C 180,E1 -5654.651,E2 -5654.651} C_VEL
LIN {X 0,Y 503.934,Z 401.713,A -85,B 0,C 180,E1 -5655.874,E2 -5655.874} C_VEL
LIN {X 0,Y 503.464,Z 411.362,A -85,B 0,C 180,E1 -5657.094,E2 -5657.094} C_VEL
LIN {X 0,Y 503.039,Z 420.969,A -85,B 0,C 180,E1 -5658.542,E2 -5658.542} C_VEL
LIN {X 0,Y 502.66,Z 429.687,A -85,B 0,C 180,E1 -5660.138,E2 -5660.138} C_VEL
LIN {X 0,Y 502.461,Z 436.033,A -85,B 0,C 180,E1 -5661.555,E2 -5661.555} C_VEL
LIN {X 0,Y 502.26,Z 441.987,A -85,B 0,C 180,E1 -5663.21,E2 -5663.21} C_VEL
LIN {X 0,Y 502.262,Z 445.313,A -85,B 0,C 180,E1 -5664.379,E2 -5664.379} C_VEL
LIN {X 0,Y 502.163,Z 448.815,A -85,B 0,C 180,E1 -5665.987,E2 -5665.987} C_VEL
LIN {X 0,Y 502.118,Z 451.134,A -85,B 0,C 180,E1 -5667.593,E2 -5667.593} C_VEL
LIN {X 0,Y 501.988,Z 452.324,A -85,B 0,C 180,E1 -5669.198,E2 -5669.198} C_VEL
LIN {X 0,Y 501.988,Z 452.343,A -85,B 0,C 180,E1 -5670.802,E2 -5670.802} C_VEL
LIN {X 0,Y 502.118,Z 451.227,A -85,B 0,C 180,E1 -5672.407,E2 -5672.407} C_VEL
LIN {X 0,Y 502.163,Z 448.981,A -85,B 0,C 180,E1 -5674.013,E2 -5674.013} C_VEL
LIN {X 0,Y 502.257,Z 445.548,A -85,B 0,C 180,E1 -5675.621,E2 -5675.621} C_VEL
LIN {X 0,Y 502.305,Z 440.85,A -85,B 0,C 180,E1 -5677.234,E2 -5677.234} C_VEL
LIN {X 0,Y 502.486,Z 434.759,A -85,B 0,C 180,E1 -5678.85,E2 -5678.85} C_VEL
LIN {X 0,Y 502.771,Z 427.088,A -85,B 0,C 180,E1 -5680.47,E2 -5680.47} C_VEL
LIN {X 0,Y 503.073,Z 418.802,A -85,B 0,C 180,E1 -5681.909,E2 -5681.909} C_VEL
LIN {X 0,Y 503.568,Z 409.051,A -85,B 0,C 180,E1 -5683.314,E2 -5683.314} C_VEL
LIN {X 0,Y 504.08,Z 398.943,A -85,B 0,C 180,E1 -5684.534,E2 -5684.534} C_VEL
LIN {X 0,Y 504.634,Z 387.6,A -85,B 0,C 180,E1 -5685.691,E2 -5685.691} C_VEL
LIN {X 0,Y 505.246,Z 375.098,A -85,B 0,C 180,E1 -5686.755,E2 -5686.755} C_VEL
LIN {X 0,Y 505.905,Z 361.727,A -85,B 0,C 180,E1 -5687.691,E2 -5687.691} C_VEL
LIN {X 0,Y 506.397,Z 349.239,A -85,B 0,C 180,E1 -5688.405,E2 -5688.405} C_VEL
LIN {X 0,Y 506.963,Z 334.625,A -85,B 0,C 180,E1 -5689.065,E2 -5689.065} C_VEL
LIN {X 0,Y 507.324,Z 319.67,A -85,B 0,C 180,E1 -5689.571,E2 -5689.571} C_VEL
LIN {X 0,Y 507.616,Z 304.447,A -85,B 0,C 180,E1 -5689.917,E2 -5689.917} C_VEL
LIN {X 0,Y 508.844,Z 159.119,A -85,B 0,C 180,E1 -5692.032,E2 -5692.032} C_VEL
LIN {X 0,Y 505.279,Z 142.664,A -85,B 0,C 180,E1 -5692.456,E2 -5692.456} C_VEL
LIN {X 0,Y 505.472,Z 135.939,A -85,B 0,C 180,E1 -5693.523,E2 -5693.523} C_VEL
LIN {X 0,Y 502.785,Z 123.485,A -85,B 0,C 180,E1 -5695.734,E2 -5695.734} C_VEL
LIN {X 0,Y 502.76,Z 123.484,A -85,B 0,C 180,E1 -5698.378,E2 -5698.378} C_VEL
LIN {X 0,Y 502.765,Z 123.488,A -85,B 0,C 180,E1 -5701.493,E2 -5701.493} C_VEL
LIN {X 0,Y 502.773,Z 123.48,A -85,B 0,C 180,E1 -5704.439,E2 -5704.439} C_VEL
LIN {X 0,Y 502.72,Z 123.491,A -85,B 0,C 180,E1 -5707.169,E2 -5707.169} C_VEL
LIN {X 0,Y 502.731,Z 123.482,A -85,B 0,C 180,E1 -5710.021,E2 -5710.021} C_VEL
LIN {X 0,Y 502.74,Z 123.488,A -85,B 0,C 180,E1 -5713.235,E2 -5713.235} C_VEL
LIN {X 0,Y 502.768,Z 123.48,A -85,B 0,C 180,E1 -5715.659,E2 -5715.659} C_VEL
LIN {X 0,Y 502.763,Z 123.486,A -85,B 0,C 180,E1 -5719.013,E2 -5719.013} C_VEL
LIN {X 0,Y 502.761,Z 123.477,A -85,B 0,C 180,E1 -5722.043,E2 -5722.043} C_VEL
LIN {X 0,Y 502.784,Z 123.481,A -85,B 0,C 180,E1 -5725.033,E2 -5725.033} C_VEL
LIN {X 0,Y 502.774,Z 123.475,A -85,B 0,C 180,E1 -5727.915,E2 -5727.915} C_VEL
LIN {X 0,Y 502.754,Z 123.486,A -85,B 0,C 180,E1 -5730.708,E2 -5730.708} C_VEL
LIN {X 0,Y 502.776,Z 123.477,A -85,B 0,C 180,E1 -5733.46,E2 -5733.46} C_VEL
LIN {X 0,Y 502.763,Z 123.484,A -85,B 0,C 180,E1 -5736.085,E2 -5736.085} C_VEL
LIN {X 0,Y 502.833,Z 123.471,A -85,B 0,C 180,E1 -5739.464,E2 -5739.464} C_VEL
LIN {X 0,Y 502.801,Z 123.479,A -85,B 0,C 180,E1 -5742.091,E2 -5742.091} C_VEL
LIN {X 0,Y 502.836,Z 123.471,A -85,B 0,C 180,E1 -5745.429,E2 -5745.429} C_VEL
LIN {X 0,Y 502.879,Z 123.466,A -85,B 0,C 180,E1 -5748.717,E2 -5748.717} C_VEL
LIN {X 0,Y 502.852,Z 123.475,A -85,B 0,C 180,E1 -5751.966,E2 -5751.966} C_VEL
LIN {X 0,Y 502.9,Z 123.462,A -85,B 0,C 180,E1 -5754.386,E2 -5754.386} C_VEL
LIN {X 0,Y 503.013,Z 123.455,A -85,B 0,C 180,E1 -5757.598,E2 -5757.598} C_VEL
LIN {X 0,Y 503.01,Z 123.45,A -85,B 0,C 180,E1 -5760,E2 -5760} C_VEL
LIN {X 0,Y 503.02,Z 123.448,A -85,B 0,C 180,E1 -5762.402,E2 -5762.402} C_VEL
LIN {X 0,Y 502.919,Z 123.466,A -85,B 0,C 180,E1 -5765.614,E2 -5765.614} C_VEL
LIN {X 0,Y 502.865,Z 123.468,A -85,B 0,C 180,E1 -5768.843,E2 -5768.843} C_VEL
LIN {X 0,Y 502.848,Z 123.47,A -85,B 0,C 180,E1 -5772.102,E2 -5772.102} C_VEL
LIN {X 0,Y 502.851,Z 123.475,A -85,B 0,C 180,E1 -5775.4,E2 -5775.4} C_VEL
LIN {X 0,Y 502.825,Z 123.473,A -85,B 0,C 180,E1 -5778.752,E2 -5778.752} C_VEL
LIN {X 0,Y 502.784,Z 123.48,A -85,B 0,C 180,E1 -5781.311,E2 -5781.311} C_VEL
LIN {X 0,Y 502.768,Z 123.48,A -85,B 0,C 180,E1 -5783.915,E2 -5783.915} C_VEL
LIN {X 0,Y 502.837,Z 123.473,A -85,B 0,C 180,E1 -5786.568,E2 -5786.568} C_VEL
LIN {X 0,Y 502.816,Z 123.473,A -85,B 0,C 180,E1 -5789.935,E2 -5789.935} C_VEL
LIN {X 0,Y 502.831,Z 123.472,A -85,B 0,C 180,E1 -5793.031,E2 -5793.031} C_VEL
LIN {X 0,Y 502.775,Z 123.479,A -85,B 0,C 180,E1 -5795.951,E2 -5795.951} C_VEL
LIN {X 0,Y 502.802,Z 123.476,A -85,B 0,C 180,E1 -5798.976,E2 -5798.976} C_VEL
LIN {X 0,Y 502.797,Z 123.48,A -85,B 0,C 180,E1 -5802.139,E2 -5802.139} C_VEL
LIN {X 0,Y 502.787,Z 123.477,A -85,B 0,C 180,E1 -5805.47,E2 -5805.47} C_VEL
LIN {X 0,Y 502.821,Z 123.47,A -85,B 0,C 180,E1 -5808.934,E2 -5808.934} C_VEL
LIN {X 0,Y 502.794,Z 123.481,A -85,B 0,C 180,E1 -5812.046,E2 -5812.046} C_VEL
LIN {X 0,Y 502.8,Z 123.476,A -85,B 0,C 180,E1 -5815.034,E2 -5815.034} C_VEL
LIN {X 0,Y 502.784,Z 123.484,A -85,B 0,C 180,E1 -5817.915,E2 -5817.915} C_VEL
LIN {X 0,Y 502.873,Z 123.546,A -85,B 0,C 180,E1 -5821.189,E2 -5821.189} C_VEL
LIN {X 0,Y 506.214,Z 137.972,A -85,B 0,C 180,E1 -5823.439,E2 -5823.439} C_VEL
LIN {X 0,Y 505.737,Z 153.44,A -85,B 0,C 180,E1 -5825.58,E2 -5825.58} C_VEL
LIN {X 0,Y 505.167,Z 168.045,A -85,B 0,C 180,E1 -5827.575,E2 -5827.575} C_VEL
LIN {X 0,Y 508.703,Z 186.772,A -85,B 0,C 180,E1 -5828.025,E2 -5828.025} C_VEL
LIN {X 0,Y 507.434,Z 334.371,A -85,B 0,C 180,E1 -5830.177,E2 -5830.177} C_VEL
LIN {X 0,Y 507.065,Z 350.12,A -85,B 0,C 180,E1 -5830.571,E2 -5830.571} C_VEL
LIN {X 0,Y 506.618,Z 364.724,A -85,B 0,C 180,E1 -5831.098,E2 -5831.098} C_VEL
LIN {X 0,Y 505.999,Z 379.273,A -85,B 0,C 180,E1 -5831.789,E2 -5831.789} C_VEL
LIN {X 0,Y 505.402,Z 392.789,A -85,B 0,C 180,E1 -5832.604,E2 -5832.604} C_VEL
LIN {X 0,Y 504.819,Z 405.255,A -85,B 0,C 180,E1 -5833.521,E2 -5833.521} C_VEL
LIN {X 0,Y 504.242,Z 417.936,A -85,B 0,C 180,E1 -5834.644,E2 -5834.644} C_VEL
LIN {X 0,Y 503.634,Z 429.457,A -85,B 0,C 180,E1 -5835.865,E2 -5835.865} C_VEL
LIN {X 0,Y 503.192,Z 439.157,A -85,B 0,C 180,E1 -5837.087,E2 -5837.087} C_VEL
LIN {X 0,Y 502.799,Z 448.853,A -85,B 0,C 180,E1 -5838.538,E2 -5838.538} C_VEL
LIN {X 0,Y 502.523,Z 456.626,A -85,B 0,C 180,E1 -5839.932,E2 -5839.932} C_VEL
LIN {X 0,Y 502.323,Z 464.04,A -85,B 0,C 180,E1 -5841.552,E2 -5841.552} C_VEL
LIN {X 0,Y 502.222,Z 469.923,A -85,B 0,C 180,E1 -5843.169,E2 -5843.169} C_VEL
LIN {X 0,Y 502.175,Z 473.418,A -85,B 0,C 180,E1 -5844.378,E2 -5844.378} C_VEL
LIN {X 0,Y 502.069,Z 476.949,A -85,B 0,C 180,E1 -5845.987,E2 -5845.987} C_VEL
LIN {X 0,Y 502.088,Z 479.274,A -85,B 0,C 180,E1 -5847.593,E2 -5847.593} C_VEL
LIN {X 0,Y 501.987,Z 480.441,A -85,B 0,C 180,E1 -5849.198,E2 -5849.198} C_VEL
LIN {X 0,Y 501.987,Z 480.44,A -85,B 0,C 180,E1 -5850.802,E2 -5850.802} C_VEL
LIN {X 0,Y 502.088,Z 479.27,A -85,B 0,C 180,E1 -5852.407,E2 -5852.407} C_VEL
LIN {X 0,Y 502.069,Z 476.944,A -85,B 0,C 180,E1 -5854.013,E2 -5854.013} C_VEL
LIN {X 0,Y 502.176,Z 473.419,A -85,B 0,C 180,E1 -5855.622,E2 -5855.622} C_VEL
LIN {X 0,Y 502.238,Z 468.599,A -85,B 0,C 180,E1 -5857.235,E2 -5857.235} C_VEL
LIN {X 0,Y 502.363,Z 462.356,A -85,B 0,C 180,E1 -5858.852,E2 -5858.852} C_VEL
LIN {X 0,Y 502.634,Z 454.519,A -85,B 0,C 180,E1 -5860.473,E2 -5860.473} C_VEL
LIN {X 0,Y 502.901,Z 445.661,A -85,B 0,C 180,E1 -5861.974,E2 -5861.974} C_VEL
LIN {X 0,Y 503.359,Z 436.143,A -85,B 0,C 180,E1 -5863.319,E2 -5863.319} C_VEL
LIN {X 0,Y 503.805,Z 425.874,A -85,B 0,C 180,E1 -5864.542,E2 -5864.542} C_VEL
LIN {X 0,Y 504.4,Z 413.813,A -85,B 0,C 180,E1 -5865.75,E2 -5865.75} C_VEL
LIN {X 0,Y 504.992,Z 401.373,A -85,B 0,C 180,E1 -5866.785,E2 -5866.785} C_VEL
LIN {X 0,Y 505.68,Z 388.025,A -85,B 0,C 180,E1 -5867.699,E2 -5867.699} C_VEL
LIN {X 0,Y 506.161,Z 375.284,A -85,B 0,C 180,E1 -5868.414,E2 -5868.414} C_VEL
LIN {X 0,Y 506.735,Z 360.948,A -85,B 0,C 180,E1 -5869.05,E2 -5869.05} C_VEL
LIN {X 0,Y 507.141,Z 345.858,A -85,B 0,C 180,E1 -5869.55,E2 -5869.55} C_VEL
LIN {X 0,Y 507.466,Z 331.083,A -85,B 0,C 180,E1 -5869.879,E2 -5869.879} C_VEL
LIN {X 0,Y 508.692,Z 186.574,A -85,B 0,C 180,E1 -5871.978,E2 -5871.978} C_VEL
LIN {X 0,Y 505.146,Z 168.067,A -85,B 0,C 180,E1 -5872.421,E2 -5872.421} C_VEL
LIN {X 0,Y 506.086,Z 145.569,A -85,B 0,C 180,E1 -5875.499,E2 -5875.499} C_VEL
LIN {X 0,Y 506.212,Z 137.964,A -85,B 0,C 180,E1 -5876.561,E2 -5876.561} C_VEL
LIN {X 0,Y 502.837,Z 123.476,A -85,B 0,C 180,E1 -5878.829,E2 -5878.829} C_VEL
LIN {X 0,Y 502.784,Z 123.48,A -85,B 0,C 180,E1 -5882.085,E2 -5882.085} C_VEL
LIN {X 0,Y 502.8,Z 123.475,A -85,B 0,C 180,E1 -5884.966,E2 -5884.966} C_VEL
LIN {X 0,Y 502.794,Z 123.483,A -85,B 0,C 180,E1 -5887.954,E2 -5887.954} C_VEL
LIN {X 0,Y 502.82,Z 123.473,A -85,B 0,C 180,E1 -5891.066,E2 -5891.066} C_VEL
LIN {X 0,Y 502.787,Z 123.476,A -85,B 0,C 180,E1 -5894.53,E2 -5894.53} C_VEL
LIN {X 0,Y 502.796,Z 123.48,A -85,B 0,C 180,E1 -5897.861,E2 -5897.861} C_VEL
LIN {X 0,Y 502.802,Z 123.477,A -85,B 0,C 180,E1 -5901.024,E2 -5901.024} C_VEL
LIN {X 0,Y 502.776,Z 123.476,A -85,B 0,C 180,E1 -5904.169,E2 -5904.169} C_VEL
LIN {X 0,Y 502.832,Z 123.473,A -85,B 0,C 180,E1 -5906.994,E2 -5906.994} C_VEL
LIN {X 0,Y 502.816,Z 123.471,A -85,B 0,C 180,E1 -5910.065,E2 -5910.065} C_VEL
LIN {X 0,Y 502.819,Z 123.473,A -85,B 0,C 180,E1 -5912.532,E2 -5912.532} C_VEL
LIN {X 0,Y 502.772,Z 123.482,A -85,B 0,C 180,E1 -5915.313,E2 -5915.313} C_VEL
LIN {X 0,Y 502.781,Z 123.478,A -85,B 0,C 180,E1 -5917.827,E2 -5917.827} C_VEL
LIN {X 0,Y 502.821,Z 123.471,A -85,B 0,C 180,E1 -5920.4,E2 -5920.4} C_VEL
LIN {X 0,Y 502.813,Z 123.478,A -85,B 0,C 180,E1 -5922.931,E2 -5922.931} C_VEL
LIN {X 0,Y 502.841,Z 123.471,A -85,B 0,C 180,E1 -5925.429,E2 -5925.429} C_VEL
LIN {X 0,Y 502.879,Z 123.471,A -85,B 0,C 180,E1 -5928.717,E2 -5928.717} C_VEL
LIN {X 0,Y 502.874,Z 123.463,A -85,B 0,C 180,E1 -5931.966,E2 -5931.966} C_VEL
LIN {X 0,Y 502.92,Z 123.466,A -85,B 0,C 180,E1 -5934.386,E2 -5934.386} C_VEL
LIN {X 0,Y 503.021,Z 123.447,A -85,B 0,C 180,E1 -5937.598,E2 -5937.598} C_VEL
LIN {X 0,Y 502.992,Z 123.453,A -85,B 0,C 180,E1 -5940.801,E2 -5940.801} C_VEL
LIN {X 0,Y 503.014,Z 123.455,A -85,B 0,C 180,E1 -5942.402,E2 -5942.402} C_VEL
LIN {X 0,Y 502.917,Z 123.46,A -85,B 0,C 180,E1 -5945.614,E2 -5945.614} C_VEL
LIN {X 0,Y 502.854,Z 123.466,A -85,B 0,C 180,E1 -5948.844,E2 -5948.844} C_VEL
LIN {X 0,Y 502.847,Z 123.474,A -85,B 0,C 180,E1 -5952.102,E2 -5952.102} C_VEL
LIN {X 0,Y 502.848,Z 123.471,A -85,B 0,C 180,E1 -5955.4,E2 -5955.4} C_VEL
LIN {X 0,Y 502.809,Z 123.474,A -85,B 0,C 180,E1 -5958.753,E2 -5958.753} C_VEL
LIN {X 0,Y 502.78,Z 123.478,A -85,B 0,C 180,E1 -5961.311,E2 -5961.311} C_VEL
LIN {X 0,Y 502.768,Z 123.482,A -85,B 0,C 180,E1 -5963.915,E2 -5963.915} C_VEL
LIN {X 0,Y 502.785,Z 123.467,A -85,B 0,C 180,E1 -5966.571,E2 -5966.571} C_VEL
LIN {X 0,Y 502.811,Z 123.477,A -85,B 0,C 180,E1 -5969.934,E2 -5969.934} C_VEL
LIN {X 0,Y 502.804,Z 123.477,A -85,B 0,C 180,E1 -5973.033,E2 -5973.033} C_VEL
LIN {X 0,Y 502.764,Z 123.48,A -85,B 0,C 180,E1 -5975.952,E2 -5975.952} C_VEL
LIN {X 0,Y 502.785,Z 123.48,A -85,B 0,C 180,E1 -5978.978,E2 -5978.978} C_VEL
LIN {X 0,Y 502.745,Z 123.48,A -85,B 0,C 180,E1 -5982.192,E2 -5982.192} C_VEL
LIN {X 0,Y 502.787,Z 123.48,A -85,B 0,C 180,E1 -5985.47,E2 -5985.47} C_VEL
LIN {X 0,Y 502.762,Z 123.486,A -85,B 0,C 180,E1 -5988.928,E2 -5988.928} C_VEL
LIN {X 0,Y 502.76,Z 123.48,A -85,B 0,C 180,E1 -5992.043,E2 -5992.043} C_VEL
LIN {X 0,Y 502.78,Z 123.484,A -85,B 0,C 180,E1 -5995.033,E2 -5995.033} C_VEL
LIN {X 0,Y 502.756,Z 123.483,A -85,B 0,C 180,E1 -5997.2,E2 -5997.2} C_VEL
LIN {X 0,Y 502.068,Z 123.569,A -85,B 0,C 180,E1 -5997.869,E2 -5997.869} C_VEL
LIN {X 0,Y 499.197,Z 123.923,A -85,B 0,C 180,E1 -5998.955,E2 -5998.955} C_VEL
LIN {X 0,Y 496.787,Z 124.219,A -85,B 0,C 180,E1 -5999.829,E2 -5999.829} C_VEL
LIN {X 0,Y 495.759,Z 124.347,A -85,B 0,C 180,E1 -6000.505,E2 -6000.505} C_VEL
LIN {X 0,Y 495.679,Z 124.359,A -85,B 0,C 180,E1 -6000.734,E2 -6000.734} C_VEL
LIN {X 0,Y 495.721,Z 124.362,A -85,B 0,C 180,E1 -6003.275,E2 -6003.275} C_VEL
LIN {X 0,Y 495.754,Z 124.476,A -85,B 0,C 180,E1 -6004.128,E2 -6004.128} C_VEL
LIN {X 0,Y 498.574,Z 137.112,A -85,B 0,C 180,E1 -6006.385,E2 -6006.385} C_VEL
LIN {X 0,Y 498.454,Z 142.902,A -85,B 0,C 180,E1 -6007.316,E2 -6007.316} C_VEL
LIN {X 0,Y 502.207,Z 159.15,A -85,B 0,C 180,E1 -6007.75,E2 -6007.75} C_VEL
LIN {X 0,Y 500.991,Z 299.363,A -85,B 0,C 180,E1 -6009.808,E2 -6009.808} C_VEL
LIN {X 0,Y 500.782,Z 315.413,A -85,B 0,C 180,E1 -6010.125,E2 -6010.125} C_VEL
LIN {X 0,Y 500.396,Z 329.877,A -85,B 0,C 180,E1 -6010.568,E2 -6010.568} C_VEL
LIN {X 0,Y 499.856,Z 344.638,A -85,B 0,C 180,E1 -6011.186,E2 -6011.186} C_VEL
LIN {X 0,Y 499.276,Z 358.874,A -85,B 0,C 180,E1 -6011.96,E2 -6011.96} C_VEL
LIN {X 0,Y 498.587,Z 372.557,A -85,B 0,C 180,E1 -6012.887,E2 -6012.887} C_VEL
LIN {X 0,Y 497.902,Z 385.602,A -85,B 0,C 180,E1 -6013.971,E2 -6013.971} C_VEL
LIN {X 0,Y 497.331,Z 396.444,A -85,B 0,C 180,E1 -6015.055,E2 -6015.055} C_VEL
LIN {X 0,Y 496.769,Z 406.94,A -85,B 0,C 180,E1 -6016.292,E2 -6016.292} C_VEL
LIN {X 0,Y 496.19,Z 417.185,A -85,B 0,C 180,E1 -6017.733,E2 -6017.733} C_VEL
LIN {X 0,Y 495.86,Z 425.687,A -85,B 0,C 180,E1 -6019.176,E2 -6019.176} C_VEL
LIN {X 0,Y 495.534,Z 432.764,A -85,B 0,C 180,E1 -6020.613,E2 -6020.613} C_VEL
LIN {X 0,Y 495.306,Z 439.328,A -85,B 0,C 180,E1 -6022.253,E2 -6022.253} C_VEL
LIN {X 0,Y 495.18,Z 444.058,A -85,B 0,C 180,E1 -6023.736,E2 -6023.736} C_VEL
LIN {X 0,Y 495.019,Z 447.42,A -85,B 0,C 180,E1 -6025.113,E2 -6025.113} C_VEL
LIN {X 0,Y 495.035,Z 450.318,A -85,B 0,C 180,E1 -6026.745,E2 -6026.745} C_VEL
LIN {X 0,Y 494.961,Z 452.067,A -85,B 0,C 180,E1 -6028.373,E2 -6028.373} C_VEL
LIN {X 0,Y 494.898,Z 452.681,A -85,B 0,C 180,E1 -6030,E2 -6030} C_VEL
LIN {X 0,Y 494.961,Z 452.122,A -85,B 0,C 180,E1 -6031.627,E2 -6031.627} C_VEL
LIN {X 0,Y 495.035,Z 450.446,A -85,B 0,C 180,E1 -6033.256,E2 -6033.256} C_VEL
LIN {X 0,Y 495.018,Z 447.618,A -85,B 0,C 180,E1 -6034.887,E2 -6034.887} C_VEL
LIN {X 0,Y 495.176,Z 444.305,A -85,B 0,C 180,E1 -6036.26,E2 -6036.26} C_VEL
LIN {X 0,Y 495.306,Z 439.635,A -85,B 0,C 180,E1 -6037.747,E2 -6037.747} C_VEL
LIN {X 0,Y 495.495,Z 433.162,A -85,B 0,C 180,E1 -6039.388,E2 -6039.388} C_VEL
LIN {X 0,Y 495.908,Z 425.066,A -85,B 0,C 180,E1 -6041.03,E2 -6041.03} C_VEL
LIN {X 0,Y 496.255,Z 416.423,A -85,B 0,C 180,E1 -6042.473,E2 -6042.473} C_VEL
LIN {X 0,Y 496.791,Z 406.022,A -85,B 0,C 180,E1 -6043.916,E2 -6043.916} C_VEL
LIN {X 0,Y 497.367,Z 395.336,A -85,B 0,C 180,E1 -6045.154,E2 -6045.154} C_VEL
LIN {X 0,Y 498.047,Z 382.972,A -85,B 0,C 180,E1 -6046.351,E2 -6046.351} C_VEL
LIN {X 0,Y 498.615,Z 370.928,A -85,B 0,C 180,E1 -6047.323,E2 -6047.323} C_VEL
LIN {X 0,Y 499.334,Z 356.864,A -85,B 0,C 180,E1 -6048.25,E2 -6048.25} C_VEL
LIN {X 0,Y 499.984,Z 342.144,A -85,B 0,C 180,E1 -6049.018,E2 -6049.018} C_VEL
LIN {X 0,Y 500.465,Z 326.824,A -85,B 0,C 180,E1 -6049.626,E2 -6049.626} C_VEL
LIN {X 0,Y 500.813,Z 311.535,A -85,B 0,C 180,E1 -6050.056,E2 -6050.056} C_VEL
LIN {X 0,Y 501.062,Z 291.749,A -85,B 0,C 180,E1 -6050.393,E2 -6050.393} C_VEL
LIN {X 0,Y 502.221,Z 159.202,A -85,B 0,C 180,E1 -6052.34,E2 -6052.34} C_VEL
LIN {X 0,Y 498.456,Z 142.863,A -85,B 0,C 180,E1 -6052.78,E2 -6052.78} C_VEL
LIN {X 0,Y 498.609,Z 137.605,A -85,B 0,C 180,E1 -6053.625,E2 -6053.625} C_VEL
LIN {X 0,Y 495.745,Z 124.361,A -85,B 0,C 180,E1 -6056.014,E2 -6056.014} C_VEL
LIN {X 0,Y 495.696,Z 124.365,A -85,B 0,C 180,E1 -6058.82,E2 -6058.82} C_VEL
LIN {X 0,Y 495.73,Z 124.362,A -85,B 0,C 180,E1 -6061.72,E2 -6061.72} C_VEL
LIN {X 0,Y 495.743,Z 124.357,A -85,B 0,C 180,E1 -6064.689,E2 -6064.689} C_VEL
LIN {X 0,Y 495.692,Z 124.367,A -85,B 0,C 180,E1 -6067.565,E2 -6067.565} C_VEL
LIN {X 0,Y 495.707,Z 124.357,A -85,B 0,C 180,E1 -6070.04,E2 -6070.04} C_VEL
LIN {X 0,Y 495.691,Z 124.367,A -85,B 0,C 180,E1 -6072.887,E2 -6072.887} C_VEL
LIN {X 0,Y 495.714,Z 124.358,A -85,B 0,C 180,E1 -6075.997,E2 -6075.997} C_VEL
LIN {X 0,Y 495.726,Z 124.359,A -85,B 0,C 180,E1 -6079.296,E2 -6079.296} C_VEL
LIN {X 0,Y 495.723,Z 124.354,A -85,B 0,C 180,E1 -6081.406,E2 -6081.406} C_VEL
LIN {X 0,Y 495.731,Z 124.357,A -85,B 0,C 180,E1 -6084.461,E2 -6084.461} C_VEL
LIN {X 0,Y 495.75,Z 124.349,A -85,B 0,C 180,E1 -6087.404,E2 -6087.404} C_VEL
LIN {X 0,Y 495.697,Z 124.358,A -85,B 0,C 180,E1 -6090.249,E2 -6090.249} C_VEL
LIN {X 0,Y 495.74,Z 124.353,A -85,B 0,C 180,E1 -6093.271,E2 -6093.271} C_VEL
LIN {X 0,Y 495.712,Z 124.359,A -85,B 0,C 180,E1 -6095.723,E2 -6095.723} C_VEL
LIN {X 0,Y 495.735,Z 124.36,A -85,B 0,C 180,E1 -6098.371,E2 -6098.371} C_VEL
LIN {X 0,Y 495.766,Z 124.35,A -85,B 0,C 180,E1 -6100.971,E2 -6100.971} C_VEL
LIN {X 0,Y 495.806,Z 124.348,A -85,B 0,C 180,E1 -6104.557,E2 -6104.557} C_VEL
LIN {X 0,Y 495.832,Z 124.35,A -85,B 0,C 180,E1 -6107.965,E2 -6107.965} C_VEL
LIN {X 0,Y 495.81,Z 124.342,A -85,B 0,C 180,E1 -6111.03,E2 -6111.03} C_VEL
LIN {X 0,Y 495.823,Z 124.348,A -85,B 0,C 180,E1 -6113.489,E2 -6113.489} C_VEL
LIN {X 0,Y 495.711,Z 124.363,A -85,B 0,C 180,E1 -6115.935,E2 -6115.935} C_VEL
LIN {X 0,Y 495.98,Z 124.33,A -85,B 0,C 180,E1 -6117.564,E2 -6117.564} C_VEL
LIN {X 0,Y 495.978,Z 124.326,A -85,B 0,C 180,E1 -6120,E2 -6120} C_VEL
LIN {X 0,Y 495.988,Z 124.324,A -85,B 0,C 180,E1 -6122.436,E2 -6122.436} C_VEL
LIN {X 0,Y 495.874,Z 124.343,A -85,B 0,C 180,E1 -6125.694,E2 -6125.694} C_VEL
LIN {X 0,Y 495.835,Z 124.344,A -85,B 0,C 180,E1 -6128.97,E2 -6128.97} C_VEL
LIN {X 0,Y 495.832,Z 124.344,A -85,B 0,C 180,E1 -6132.035,E2 -6132.035} C_VEL
LIN {X 0,Y 495.826,Z 124.35,A -85,B 0,C 180,E1 -6135.451,E2 -6135.451} C_VEL
LIN {X 0,Y 495.781,Z 124.354,A -85,B 0,C 180,E1 -6139.028,E2 -6139.028} C_VEL
LIN {X 0,Y 495.744,Z 124.354,A -85,B 0,C 180,E1 -6141.629,E2 -6141.629} C_VEL
LIN {X 0,Y 495.715,Z 124.359,A -85,B 0,C 180,E1 -6144.277,E2 -6144.277} C_VEL
LIN {X 0,Y 495.763,Z 124.357,A -85,B 0,C 180,E1 -6146.977,E2 -6146.977} C_VEL
LIN {X 0,Y 495.766,Z 124.353,A -85,B 0,C 180,E1 -6150.147,E2 -6150.147} C_VEL
LIN {X 0,Y 495.791,Z 124.347,A -85,B 0,C 180,E1 -6153.243,E2 -6153.243} C_VEL
LIN {X 0,Y 495.721,Z 124.359,A -85,B 0,C 180,E1 -6156.088,E2 -6156.088} C_VEL
LIN {X 0,Y 495.764,Z 124.355,A -85,B 0,C 180,E1 -6158.768,E2 -6158.768} C_VEL
LIN {X 0,Y 495.757,Z 124.354,A -85,B 0,C 180,E1 -6161.781,E2 -6161.781} C_VEL
LIN {X 0,Y 495.739,Z 124.355,A -85,B 0,C 180,E1 -6165.141,E2 -6165.141} C_VEL
LIN {X 0,Y 495.757,Z 124.359,A -85,B 0,C 180,E1 -6168.219,E2 -6168.219} C_VEL
LIN {X 0,Y 495.752,Z 124.354,A -85,B 0,C 180,E1 -6171.408,E2 -6171.408} C_VEL
LIN {X 0,Y 495.749,Z 124.357,A -85,B 0,C 180,E1 -6174.462,E2 -6174.462} C_VEL
LIN {X 0,Y 495.768,Z 124.355,A -85,B 0,C 180,E1 -6177.405,E2 -6177.405} C_VEL
LIN {X 0,Y 495.815,Z 124.426,A -85,B 0,C 180,E1 -6180.898,E2 -6180.898} C_VEL
LIN {X 0,Y 499.27,Z 139.086,A -85,B 0,C 180,E1 -6183.227,E2 -6183.227} C_VEL
LIN {X 0,Y 499.431,Z 142.241,A -85,B 0,C 180,E1 -6183.687,E2 -6183.687} C_VEL
LIN {X 0,Y 498.496,Z 164.221,A -85,B 0,C 180,E1 -6186.749,E2 -6186.749} C_VEL
LIN {X 0,Y 498.321,Z 167.865,A -85,B 0,C 180,E1 -6187.253,E2 -6187.253} C_VEL
LIN {X 0,Y 502.103,Z 187.95,A -85,B 0,C 180,E1 -6187.741,E2 -6187.741} C_VEL
LIN {X 0,Y 500.757,Z 334.181,A -85,B 0,C 180,E1 -6189.902,E2 -6189.902} C_VEL
LIN {X 0,Y 500.344,Z 349.925,A -85,B 0,C 180,E1 -6190.299,E2 -6190.299} C_VEL
LIN {X 0,Y 499.88,Z 364.901,A -85,B 0,C 180,E1 -6190.849,E2 -6190.849} C_VEL
LIN {X 0,Y 499.221,Z 379.076,A -85,B 0,C 180,E1 -6191.533,E2 -6191.533} C_VEL
LIN {X 0,Y 498.582,Z 392.59,A -85,B 0,C 180,E1 -6192.358,E2 -6192.358} C_VEL
LIN {X 0,Y 497.969,Z 405.056,A -85,B 0,C 180,E1 -6193.288,E2 -6193.288} C_VEL
LIN {X 0,Y 497.334,Z 417.736,A -85,B 0,C 180,E1 -6194.425,E2 -6194.425} C_VEL
LIN {X 0,Y 496.681,Z 429.256,A -85,B 0,C 180,E1 -6195.663,E2 -6195.663} C_VEL
LIN {X 0,Y 496.199,Z 438.956,A -85,B 0,C 180,E1 -6196.902,E2 -6196.902} C_VEL
LIN {X 0,Y 495.799,Z 448.375,A -85,B 0,C 180,E1 -6198.328,E2 -6198.328} C_VEL
LIN {X 0,Y 495.495,Z 456.426,A -85,B 0,C 180,E1 -6199.788,E2 -6199.788} C_VEL
LIN {X 0,Y 495.237,Z 463.839,A -85,B 0,C 180,E1 -6201.431,E2 -6201.431} C_VEL
LIN {X 0,Y 495.151,Z 469.722,A -85,B 0,C 180,E1 -6203.071,E2 -6203.071} C_VEL
LIN {X 0,Y 495.07,Z 473.218,A -85,B 0,C 180,E1 -6204.297,E2 -6204.297} C_VEL
LIN {X 0,Y 494.967,Z 476.749,A -85,B 0,C 180,E1 -6205.929,E2 -6205.929} C_VEL
LIN {X 0,Y 494.994,Z 479.075,A -85,B 0,C 180,E1 -6207.559,E2 -6207.559} C_VEL
LIN {X 0,Y 494.907,Z 480.243,A -85,B 0,C 180,E1 -6209.186,E2 -6209.186} C_VEL
LIN {X 0,Y 494.907,Z 480.242,A -85,B 0,C 180,E1 -6210.814,E2 -6210.814} C_VEL
LIN {X 0,Y 494.994,Z 479.071,A -85,B 0,C 180,E1 -6212.441,E2 -6212.441} C_VEL
LIN {X 0,Y 494.967,Z 476.745,A -85,B 0,C 180,E1 -6214.071,E2 -6214.071} C_VEL
LIN {X 0,Y 495.073,Z 473.219,A -85,B 0,C 180,E1 -6215.703,E2 -6215.703} C_VEL
LIN {X 0,Y 495.157,Z 468.399,A -85,B 0,C 180,E1 -6217.339,E2 -6217.339} C_VEL
LIN {X 0,Y 495.287,Z 462.156,A -85,B 0,C 180,E1 -6218.98,E2 -6218.98} C_VEL
LIN {X 0,Y 495.594,Z 454.318,A -85,B 0,C 180,E1 -6220.623,E2 -6220.623} C_VEL
LIN {X 0,Y 495.872,Z 446.038,A -85,B 0,C 180,E1 -6222.058,E2 -6222.058} C_VEL
LIN {X 0,Y 496.381,Z 435.942,A -85,B 0,C 180,E1 -6223.51,E2 -6223.51} C_VEL
LIN {X 0,Y 496.853,Z 425.673,A -85,B 0,C 180,E1 -6224.751,E2 -6224.751} C_VEL
LIN {X 0,Y 497.53,Z 413.267,A -85,B 0,C 180,E1 -6226.006,E2 -6226.006} C_VEL
LIN {X 0,Y 498.229,Z 399.836,A -85,B 0,C 180,E1 -6227.125,E2 -6227.125} C_VEL
LIN {X 0,Y 498.952,Z 386.195,A -85,B 0,C 180,E1 -6228.052,E2 -6228.052} C_VEL
LIN {X 0,Y 499.547,Z 372.068,A -85,B 0,C 180,E1 -6228.826,E2 -6228.826} C_VEL
LIN {X 0,Y 500.139,Z 356.756,A -85,B 0,C 180,E1 -6229.471,E2 -6229.471} C_VEL
LIN {X 0,Y 500.585,Z 341.646,A -85,B 0,C 180,E1 -6229.932,E2 -6229.932} C_VEL
LIN {X 0,Y 500.862,Z 325.743,A -85,B 0,C 180,E1 -6230.241,E2 -6230.241} C_VEL
LIN {X 0,Y 502.097,Z 188.213,A -85,B 0,C 180,E1 -6232.254,E2 -6232.254} C_VEL
LIN {X 0,Y 498.911,Z 170.947,A -85,B 0,C 180,E1 -6232.666,E2 -6232.666} C_VEL
LIN {X 0,Y 498.341,Z 167.683,A -85,B 0,C 180,E1 -6232.77,E2 -6232.77} C_VEL
LIN {X 0,Y 499.333,Z 145.378,A -85,B 0,C 180,E1 -6235.869,E2 -6235.869} C_VEL
LIN {X 0,Y 499.479,Z 140.657,A -85,B 0,C 180,E1 -6236.535,E2 -6236.535} C_VEL
LIN {X 0,Y 496.786,Z 128.445,A -85,B 0,C 180,E1 -6238.451,E2 -6238.451} C_VEL
LIN {X 0,Y 495.791,Z 124.354,A -85,B 0,C 180,E1 -6239.133,E2 -6239.133} C_VEL
LIN {X 0,Y 495.768,Z 124.348,A -85,B 0,C 180,E1 -6242.594,E2 -6242.594} C_VEL
LIN {X 0,Y 495.749,Z 124.356,A -85,B 0,C 180,E1 -6245.538,E2 -6245.538} C_VEL
LIN {X 0,Y 495.765,Z 124.352,A -85,B 0,C 180,E1 -6248.768,E2 -6248.768} C_VEL
LIN {X 0,Y 495.757,Z 124.36,A -85,B 0,C 180,E1 -6251.781,E2 -6251.781} C_VEL
LIN {X 0,Y 495.738,Z 124.356,A -85,B 0,C 180,E1 -6255.141,E2 -6255.141} C_VEL
LIN {X 0,Y 495.757,Z 124.353,A -85,B 0,C 180,E1 -6258.219,E2 -6258.219} C_VEL
LIN {X 0,Y 495.751,Z 124.358,A -85,B 0,C 180,E1 -6261.409,E2 -6261.409} C_VEL
LIN {X 0,Y 495.748,Z 124.351,A -85,B 0,C 180,E1 -6264.462,E2 -6264.462} C_VEL
LIN {X 0,Y 495.767,Z 124.356,A -85,B 0,C 180,E1 -6267.406,E2 -6267.406} C_VEL
LIN {X 0,Y 495.767,Z 124.349,A -85,B 0,C 180,E1 -6270.254,E2 -6270.254} C_VEL
LIN {X 0,Y 495.806,Z 124.351,A -85,B 0,C 180,E1 -6273.255,E2 -6273.255} C_VEL
LIN {X 0,Y 495.74,Z 124.356,A -85,B 0,C 180,E1 -6276.612,E2 -6276.612} C_VEL
LIN {X 0,Y 495.781,Z 124.35,A -85,B 0,C 180,E1 -6279.324,E2 -6279.324} C_VEL
LIN {X 0,Y 495.781,Z 124.35,A -85,B 0,C 180,E1 -6281.829,E2 -6281.829} C_VEL
LIN {X 0,Y 495.826,Z 124.345,A -85,B 0,C 180,E1 -6284.549,E2 -6284.549} C_VEL
LIN {X 0,Y 495.831,Z 124.34,A -85,B 0,C 180,E1 -6287.965,E2 -6287.965} C_VEL
LIN {X 0,Y 495.835,Z 124.342,A -85,B 0,C 180,E1 -6291.03,E2 -6291.03} C_VEL
LIN {X 0,Y 495.875,Z 124.343,A -85,B 0,C 180,E1 -6294.306,E2 -6294.306} C_VEL
LIN {X 0,Y 495.988,Z 124.323,A -85,B 0,C 180,E1 -6297.564,E2 -6297.564} C_VEL
LIN {X 0,Y 495.944,Z 124.331,A -85,B 0,C 180,E1 -6300.812,E2 -6300.812} C_VEL
LIN {X 0,Y 495.981,Z 124.331,A -85,B 0,C 180,E1 -6302.436,E2 -6302.436} C_VEL
LIN {X 0,Y 495.872,Z 124.338,A -85,B 0,C 180,E1 -6305.694,E2 -6305.694} C_VEL
LIN {X 0,Y 495.811,Z 124.343,A -85,B 0,C 180,E1 -6308.97,E2 -6308.97} C_VEL
LIN {X 0,Y 495.831,Z 124.349,A -85,B 0,C 180,E1 -6312.035,E2 -6312.035} C_VEL
LIN {X 0,Y 495.805,Z 124.348,A -85,B 0,C 180,E1 -6315.442,E2 -6315.442} C_VEL
LIN {X 0,Y 495.769,Z 124.351,A -85,B 0,C 180,E1 -6319.029,E2 -6319.029} C_VEL
LIN {X 0,Y 495.741,Z 124.358,A -85,B 0,C 180,E1 -6321.629,E2 -6321.629} C_VEL
LIN {X 0,Y 495.714,Z 124.357,A -85,B 0,C 180,E1 -6324.277,E2 -6324.277} C_VEL
LIN {X 0,Y 495.733,Z 124.346,A -85,B 0,C 180,E1 -6326.979,E2 -6326.979} C_VEL
LIN {X 0,Y 495.758,Z 124.353,A -85,B 0,C 180,E1 -6330.145,E2 -6330.145} C_VEL
LIN {X 0,Y 495.752,Z 124.358,A -85,B 0,C 180,E1 -6333.237,E2 -6333.237} C_VEL
LIN {X 0,Y 495.709,Z 124.358,A -85,B 0,C 180,E1 -6336.086,E2 -6336.086} C_VEL
LIN {X 0,Y 495.743,Z 124.355,A -85,B 0,C 180,E1 -6338.765,E2 -6338.765} C_VEL
LIN {X 0,Y 495.724,Z 124.356,A -85,B 0,C 180,E1 -6341.785,E2 -6341.785} C_VEL
LIN {X 0,Y 495.738,Z 124.361,A -85,B 0,C 180,E1 -6345.141,E2 -6345.141} C_VEL
LIN {X 0,Y 495.724,Z 124.358,A -85,B 0,C 180,E1 -6348.215,E2 -6348.215} C_VEL
LIN {X 0,Y 495.738,Z 124.357,A -85,B 0,C 180,E1 -6351.236,E2 -6351.236} C_VEL
LIN {X 0,Y 495.728,Z 124.359,A -85,B 0,C 180,E1 -6354.461,E2 -6354.461} C_VEL
LIN {X 0,Y 495.724,Z 124.36,A -85,B 0,C 180,E1 -6357.402,E2 -6357.402} C_VEL
LIN {X 0,Y 495.695,Z 124.353,A -85,B 0,C 180,E1 -6360.249,E2 -6360.249} C_VEL
LIN {X 0,Y 495.679,Z 124.359,A -85,B 0,C 180,E1 -6360.734,E2 -6360.734} C_VEL
LIN {X 0,Y 495.007,Z 124.449,A -85,B 0,C 180,E1 -6361.187,E2 -6361.187} C_VEL
LIN {X 0,Y 492.172,Z 124.804,A -85,B 0,C 180,E1 -6361.896,E2 -6361.896} C_VEL
LIN {X 0,Y 489.337,Z 125.157,A -85,B 0,C 180,E1 -6362.612,E2 -6362.612} C_VEL
LIN {X 0,Y 488.684,Z 125.241,A -85,B 0,C 180,E1 -6363.074,E2 -6363.074} C_VEL
LIN {X 0,Y 488.689,Z 125.328,A -85,B 0,C 180,E1 -6363.84,E2 -6363.84} C_VEL
LIN {X 0,Y 491.807,Z 139.561,A -85,B 0,C 180,E1 -6366.414,E2 -6366.414} C_VEL
LIN {X 0,Y 491.711,Z 143.395,A -85,B 0,C 180,E1 -6366.998,E2 -6366.998} C_VEL
LIN {X 0,Y 495.702,Z 160.699,A -85,B 0,C 180,E1 -6367.462,E2 -6367.462} C_VEL
LIN {X 0,Y 494.267,Z 308.446,A -85,B 0,C 180,E1 -6369.68,E2 -6369.68} C_VEL
LIN {X 0,Y 493.873,Z 323.959,A -85,B 0,C 180,E1 -6370.082,E2 -6370.082} C_VEL
LIN {X 0,Y 493.417,Z 339.334,A -85,B 0,C 180,E1 -6370.666,E2 -6370.666} C_VEL
LIN {X 0,Y 492.884,Z 351.904,A -85,B 0,C 180,E1 -6371.287,E2 -6371.287} C_VEL
LIN {X 0,Y 492.174,Z 365.504,A -85,B 0,C 180,E1 -6372.121,E2 -6372.121} C_VEL
LIN {X 0,Y 491.531,Z 378.002,A -85,B 0,C 180,E1 -6373.063,E2 -6373.063} C_VEL
LIN {X 0,Y 490.88,Z 389.111,A -85,B 0,C 180,E1 -6374.06,E2 -6374.06} C_VEL
LIN {X 0,Y 490.224,Z 400.351,A -85,B 0,C 180,E1 -6375.258,E2 -6375.258} C_VEL
LIN {X 0,Y 489.645,Z 410.294,A -85,B 0,C 180,E1 -6376.512,E2 -6376.512} C_VEL
LIN {X 0,Y 489.101,Z 419.459,A -85,B 0,C 180,E1 -6377.881,E2 -6377.881} C_VEL
LIN {X 0,Y 488.698,Z 428.091,A -85,B 0,C 180,E1 -6379.435,E2 -6379.435} C_VEL
LIN {X 0,Y 488.436,Z 434.761,A -85,B 0,C 180,E1 -6380.893,E2 -6380.893} C_VEL
LIN {X 0,Y 488.178,Z 440.943,A -85,B 0,C 180,E1 -6382.555,E2 -6382.555} C_VEL
LIN {X 0,Y 488.134,Z 445.714,A -85,B 0,C 180,E1 -6384.216,E2 -6384.216} C_VEL
LIN {X 0,Y 487.964,Z 449.216,A -85,B 0,C 180,E1 -6385.87,E2 -6385.87} C_VEL
LIN {X 0,Y 487.929,Z 451.533,A -85,B 0,C 180,E1 -6387.523,E2 -6387.523} C_VEL
LIN {X 0,Y 487.831,Z 452.721,A -85,B 0,C 180,E1 -6389.175,E2 -6389.175} C_VEL
LIN {X 0,Y 487.832,Z 452.739,A -85,B 0,C 180,E1 -6390.826,E2 -6390.826} C_VEL
LIN {X 0,Y 487.93,Z 451.623,A -85,B 0,C 180,E1 -6392.477,E2 -6392.477} C_VEL
LIN {X 0,Y 487.963,Z 449.377,A -85,B 0,C 180,E1 -6394.13,E2 -6394.13} C_VEL
LIN {X 0,Y 488.106,Z 445.943,A -85,B 0,C 180,E1 -6395.785,E2 -6395.785} C_VEL
LIN {X 0,Y 488.177,Z 441.244,A -85,B 0,C 180,E1 -6397.445,E2 -6397.445} C_VEL
LIN {X 0,Y 488.417,Z 435.152,A -85,B 0,C 180,E1 -6399.107,E2 -6399.107} C_VEL
LIN {X 0,Y 488.777,Z 427.48,A -85,B 0,C 180,E1 -6400.773,E2 -6400.773} C_VEL
LIN {X 0,Y 489.188,Z 418.7,A -85,B 0,C 180,E1 -6402.33,E2 -6402.33} C_VEL
LIN {X 0,Y 489.678,Z 409.443,A -85,B 0,C 180,E1 -6403.699,E2 -6403.699} C_VEL
LIN {X 0,Y 490.287,Z 399.333,A -85,B 0,C 180,E1 -6404.953,E2 -6404.953} C_VEL
LIN {X 0,Y 490.918,Z 388.527,A -85,B 0,C 180,E1 -6406.087,E2 -6406.087} C_VEL
LIN {X 0,Y 491.579,Z 376.512,A -85,B 0,C 180,E1 -6407.15,E2 -6407.15} C_VEL
LIN {X 0,Y 492.296,Z 363.686,A -85,B 0,C 180,E1 -6408.09,E2 -6408.09} C_VEL
LIN {X 0,Y 492.945,Z 349.618,A -85,B 0,C 180,E1 -6408.926,E2 -6408.926} C_VEL
LIN {X 0,Y 493.564,Z 334.528,A -85,B 0,C 180,E1 -6409.624,E2 -6409.624} C_VEL
LIN {X 0,Y 493.969,Z 319.663,A -85,B 0,C 180,E1 -6410.134,E2 -6410.134} C_VEL
LIN {X 0,Y 494.314,Z 303.831,A -85,B 0,C 180,E1 -6410.494,E2 -6410.494} C_VEL
LIN {X 0,Y 495.638,Z 160.162,A -85,B 0,C 180,E1 -6412.64,E2 -6412.64} C_VEL
LIN {X 0,Y 491.676,Z 143.071,A -85,B 0,C 180,E1 -6413.109,E2 -6413.109} C_VEL
LIN {X 0,Y 491.674,Z 138.754,A -85,B 0,C 180,E1 -6413.82,E2 -6413.82} C_VEL
LIN {X 0,Y 488.682,Z 125.241,A -85,B 0,C 180,E1 -6416.304,E2 -6416.304} C_VEL
LIN {X 0,Y 488.66,Z 125.244,A -85,B 0,C 180,E1 -6419.275,E2 -6419.275} C_VEL
LIN {X 0,Y 488.679,Z 125.237,A -85,B 0,C 180,E1 -6422.149,E2 -6422.149} C_VEL
LIN {X 0,Y 488.698,Z 125.24,A -85,B 0,C 180,E1 -6425.117,E2 -6425.117} C_VEL
LIN {X 0,Y 488.645,Z 125.241,A -85,B 0,C 180,E1 -6428.203,E2 -6428.203} C_VEL
LIN {X 0,Y 488.644,Z 125.243,A -85,B 0,C 180,E1 -6431.422,E2 -6431.422} C_VEL
LIN {X 0,Y 488.697,Z 125.237,A -85,B 0,C 180,E1 -6434.804,E2 -6434.804} C_VEL
LIN {X 0,Y 488.649,Z 125.233,A -85,B 0,C 180,E1 -6437.47,E2 -6437.47} C_VEL
LIN {X 0,Y 488.705,Z 125.232,A -85,B 0,C 180,E1 -6439.674,E2 -6439.674} C_VEL
LIN {X 0,Y 488.652,Z 125.235,A -85,B 0,C 180,E1 -6442.839,E2 -6442.839} C_VEL
LIN {X 0,Y 488.718,Z 125.23,A -85,B 0,C 180,E1 -6445.886,E2 -6445.886} C_VEL
LIN {X 0,Y 488.664,Z 125.231,A -85,B 0,C 180,E1 -6448.818,E2 -6448.818} C_VEL
LIN {X 0,Y 488.686,Z 125.233,A -85,B 0,C 180,E1 -6451.667,E2 -6451.667} C_VEL
LIN {X 0,Y 488.692,Z 125.237,A -85,B 0,C 180,E1 -6454.441,E2 -6454.441} C_VEL
LIN {X 0,Y 488.709,Z 125.229,A -85,B 0,C 180,E1 -6457.152,E2 -6457.152} C_VEL
LIN {X 0,Y 488.719,Z 125.232,A -85,B 0,C 180,E1 -6459.81,E2 -6459.81} C_VEL
LIN {X 0,Y 488.68,Z 125.238,A -85,B 0,C 180,E1 -6462.421,E2 -6462.421} C_VEL
LIN {X 0,Y 488.753,Z 125.224,A -85,B 0,C 180,E1 -6464.999,E2 -6464.999} C_VEL
LIN {X 0,Y 488.808,Z 125.221,A -85,B 0,C 180,E1 -6468.388,E2 -6468.388} C_VEL
LIN {X 0,Y 488.764,Z 125.225,A -85,B 0,C 180,E1 -6471.733,E2 -6471.733} C_VEL
LIN {X 0,Y 488.817,Z 125.217,A -85,B 0,C 180,E1 -6474.224,E2 -6474.224} C_VEL
LIN {X 0,Y 488.946,Z 125.206,A -85,B 0,C 180,E1 -6477.528,E2 -6477.528} C_VEL
LIN {X 0,Y 488.947,Z 125.201,A -85,B 0,C 180,E1 -6480,E2 -6480} C_VEL
LIN {X 0,Y 488.955,Z 125.2,A -85,B 0,C 180,E1 -6482.471,E2 -6482.471} C_VEL
LIN {X 0,Y 488.832,Z 125.219,A -85,B 0,C 180,E1 -6485.776,E2 -6485.776} C_VEL
LIN {X 0,Y 488.783,Z 125.22,A -85,B 0,C 180,E1 -6488.267,E2 -6488.267} C_VEL
LIN {X 0,Y 488.808,Z 125.223,A -85,B 0,C 180,E1 -6491.612,E2 -6491.612} C_VEL
LIN {X 0,Y 488.757,Z 125.228,A -85,B 0,C 180,E1 -6495,E2 -6495} C_VEL
LIN {X 0,Y 488.748,Z 125.223,A -85,B 0,C 180,E1 -6498.442,E2 -6498.442} C_VEL
LIN {X 0,Y 488.709,Z 125.237,A -85,B 0,C 180,E1 -6501.071,E2 -6501.071} C_VEL
LIN {X 0,Y 488.671,Z 125.236,A -85,B 0,C 180,E1 -6503.746,E2 -6503.746} C_VEL
LIN {X 0,Y 488.727,Z 125.233,A -85,B 0,C 180,E1 -6506.928,E2 -6506.928} C_VEL
LIN {X 0,Y 488.725,Z 125.231,A -85,B 0,C 180,E1 -6510.219,E2 -6510.219} C_VEL
LIN {X 0,Y 488.731,Z 125.225,A -85,B 0,C 180,E1 -6513.483,E2 -6513.483} C_VEL
LIN {X 0,Y 488.684,Z 125.239,A -85,B 0,C 180,E1 -6516.354,E2 -6516.354} C_VEL
LIN {X 0,Y 488.702,Z 125.231,A -85,B 0,C 180,E1 -6519.254,E2 -6519.254} C_VEL
LIN {X 0,Y 488.708,Z 125.231,A -85,B 0,C 180,E1 -6521.599,E2 -6521.599} C_VEL
LIN {X 0,Y 488.703,Z 125.234,A -85,B 0,C 180,E1 -6524.802,E2 -6524.802} C_VEL
LIN {X 0,Y 488.693,Z 125.232,A -85,B 0,C 180,E1 -6527.474,E2 -6527.474} C_VEL
LIN {X 0,Y 488.734,Z 125.226,A -85,B 0,C 180,E1 -6529.676,E2 -6529.676} C_VEL
LIN {X 0,Y 488.68,Z 125.235,A -85,B 0,C 180,E1 -6532.841,E2 -6532.841} C_VEL
LIN {X 0,Y 488.731,Z 125.235,A -85,B 0,C 180,E1 -6535.887,E2 -6535.887} C_VEL
LIN {X 0,Y 488.693,Z 125.235,A -85,B 0,C 180,E1 -6538.82,E2 -6538.82} C_VEL
LIN {X 0,Y 488.76,Z 125.419,A -85,B 0,C 180,E1 -6540.614,E2 -6540.614} C_VEL
LIN {X 0,Y 492.013,Z 138.889,A -85,B 0,C 180,E1 -6542.8,E2 -6542.8} C_VEL
LIN {X 0,Y 492.659,Z 142.054,A -85,B 0,C 180,E1 -6543.297,E2 -6543.297} C_VEL
LIN {X 0,Y 491.789,Z 162.182,A -85,B 0,C 180,E1 -6546.149,E2 -6546.149} C_VEL
LIN {X 0,Y 491.51,Z 167.643,A -85,B 0,C 180,E1 -6546.917,E2 -6546.917} C_VEL
LIN {X 0,Y 495.532,Z 189.186,A -85,B 0,C 180,E1 -6547.452,E2 -6547.452} C_VEL
LIN {X 0,Y 494.073,Z 334.628,A -85,B 0,C 180,E1 -6549.632,E2 -6549.632} C_VEL
LIN {X 0,Y 493.624,Z 350.406,A -85,B 0,C 180,E1 -6550.043,E2 -6550.043} C_VEL
LIN {X 0,Y 493.144,Z 365.084,A -85,B 0,C 180,E1 -6550.595,E2 -6550.595} C_VEL
LIN {X 0,Y 492.46,Z 378.879,A -85,B 0,C 180,E1 -6551.27,E2 -6551.27} C_VEL
LIN {X 0,Y 491.781,Z 392.393,A -85,B 0,C 180,E1 -6552.106,E2 -6552.106} C_VEL
LIN {X 0,Y 491.042,Z 406.153,A -85,B 0,C 180,E1 -6553.152,E2 -6553.152} C_VEL
LIN {X 0,Y 490.386,Z 418.611,A -85,B 0,C 180,E1 -6554.305,E2 -6554.305} C_VEL
LIN {X 0,Y 489.714,Z 429.056,A -85,B 0,C 180,E1 -6555.455,E2 -6555.455} C_VEL
LIN {X 0,Y 489.23,Z 438.756,A -85,B 0,C 180,E1 -6556.712,E2 -6556.712} C_VEL
LIN {X 0,Y 488.775,Z 448.456,A -85,B 0,C 180,E1 -6558.205,E2 -6558.205} C_VEL
LIN {X 0,Y 488.465,Z 456.226,A -85,B 0,C 180,E1 -6559.639,E2 -6559.639} C_VEL
LIN {X 0,Y 488.159,Z 463.638,A -85,B 0,C 180,E1 -6561.305,E2 -6561.305} C_VEL
LIN {X 0,Y 488.066,Z 469.522,A -85,B 0,C 180,E1 -6562.969,E2 -6562.969} C_VEL
LIN {X 0,Y 487.97,Z 473.018,A -85,B 0,C 180,E1 -6564.214,E2 -6564.214} C_VEL
LIN {X 0,Y 487.868,Z 476.55,A -85,B 0,C 180,E1 -6565.869,E2 -6565.869} C_VEL
LIN {X 0,Y 487.904,Z 478.877,A -85,B 0,C 180,E1 -6567.523,E2 -6567.523} C_VEL
LIN {X 0,Y 487.83,Z 480.045,A -85,B 0,C 180,E1 -6569.174,E2 -6569.174} C_VEL
LIN {X 0,Y 487.83,Z 480.044,A -85,B 0,C 180,E1 -6570.825,E2 -6570.825} C_VEL
LIN {X 0,Y 487.904,Z 478.873,A -85,B 0,C 180,E1 -6572.477,E2 -6572.477} C_VEL
LIN {X 0,Y 487.868,Z 476.546,A -85,B 0,C 180,E1 -6574.13,E2 -6574.13} C_VEL
LIN {X 0,Y 487.975,Z 473.02,A -85,B 0,C 180,E1 -6575.786,E2 -6575.786} C_VEL
LIN {X 0,Y 488.06,Z 468.199,A -85,B 0,C 180,E1 -6577.446,E2 -6577.446} C_VEL
LIN {X 0,Y 488.222,Z 461.956,A -85,B 0,C 180,E1 -6579.111,E2 -6579.111} C_VEL
LIN {X 0,Y 488.567,Z 454.118,A -85,B 0,C 180,E1 -6580.778,E2 -6580.778} C_VEL
LIN {X 0,Y 488.842,Z 445.981,A -85,B 0,C 180,E1 -6582.211,E2 -6582.211} C_VEL
LIN {X 0,Y 489.411,Z 435.741,A -85,B 0,C 180,E1 -6583.706,E2 -6583.706} C_VEL
LIN {X 0,Y 489.911,Z 425.471,A -85,B 0,C 180,E1 -6584.964,E2 -6584.964} C_VEL
LIN {X 0,Y 490.642,Z 413.065,A -85,B 0,C 180,E1 -6586.237,E2 -6586.237} C_VEL
LIN {X 0,Y 491.369,Z 399.632,A -85,B 0,C 180,E1 -6587.372,E2 -6587.372} C_VEL
LIN {X 0,Y 492.156,Z 385.992,A -85,B 0,C 180,E1 -6588.31,E2 -6588.31} C_VEL
LIN {X 0,Y 492.803,Z 371.865,A -85,B 0,C 180,E1 -6589.094,E2 -6589.094} C_VEL
LIN {X 0,Y 493.447,Z 356.434,A -85,B 0,C 180,E1 -6589.75,E2 -6589.75} C_VEL
LIN {X 0,Y 493.904,Z 340.988,A -85,B 0,C 180,E1 -6590.224,E2 -6590.224} C_VEL
LIN {X 0,Y 494.214,Z 325.55,A -85,B 0,C 180,E1 -6590.525,E2 -6590.525} C_VEL
LIN {X 0,Y 495.521,Z 189.125,A -85,B 0,C 180,E1 -6592.548,E2 -6592.548} C_VEL
LIN {X 0,Y 491.857,Z 169.563,A -85,B 0,C 180,E1 -6593.027,E2 -6593.027} C_VEL
LIN {X 0,Y 491.522,Z 167.479,A -85,B 0,C 180,E1 -6593.104,E2 -6593.104} C_VEL
LIN {X 0,Y 492.532,Z 146.185,A -85,B 0,C 180,E1 -6596.109,E2 -6596.109} C_VEL
LIN {X 0,Y 492.612,Z 142.04,A -85,B 0,C 180,E1 -6596.706,E2 -6596.706} C_VEL
LIN {X 0,Y 489.847,Z 129.738,A -85,B 0,C 180,E1 -6598.671,E2 -6598.671} C_VEL
LIN {X 0,Y 488.73,Z 125.233,A -85,B 0,C 180,E1 -6599.447,E2 -6599.447} C_VEL
LIN {X 0,Y 488.704,Z 125.232,A -85,B 0,C 180,E1 -6602.147,E2 -6602.147} C_VEL
LIN {X 0,Y 488.718,Z 125.229,A -85,B 0,C 180,E1 -6605.115,E2 -6605.115} C_VEL
LIN {X 0,Y 488.681,Z 125.239,A -85,B 0,C 180,E1 -6608.2,E2 -6608.2} C_VEL
LIN {X 0,Y 488.719,Z 125.231,A -85,B 0,C 180,E1 -6610.345,E2 -6610.345} C_VEL
LIN {X 0,Y 488.686,Z 125.241,A -85,B 0,C 180,E1 -6613.655,E2 -6613.655} C_VEL
LIN {X 0,Y 488.686,Z 125.233,A -85,B 0,C 180,E1 -6616.346,E2 -6616.346} C_VEL
LIN {X 0,Y 488.734,Z 125.233,A -85,B 0,C 180,E1 -6619.677,E2 -6619.677} C_VEL
LIN {X 0,Y 488.68,Z 125.234,A -85,B 0,C 180,E1 -6622.841,E2 -6622.841} C_VEL
LIN {X 0,Y 488.725,Z 125.229,A -85,B 0,C 180,E1 -6625.887,E2 -6625.887} C_VEL
LIN {X 0,Y 488.693,Z 125.234,A -85,B 0,C 180,E1 -6628.82,E2 -6628.82} C_VEL
LIN {X 0,Y 488.742,Z 125.228,A -85,B 0,C 180,E1 -6631.671,E2 -6631.671} C_VEL
LIN {X 0,Y 488.706,Z 125.231,A -85,B 0,C 180,E1 -6634.442,E2 -6634.442} C_VEL
LIN {X 0,Y 488.723,Z 125.235,A -85,B 0,C 180,E1 -6637.153,E2 -6637.153} C_VEL
LIN {X 0,Y 488.725,Z 125.226,A -85,B 0,C 180,E1 -6639.811,E2 -6639.811} C_VEL
LIN {X 0,Y 488.711,Z 125.233,A -85,B 0,C 180,E1 -6642.423,E2 -6642.423} C_VEL
LIN {X 0,Y 488.762,Z 125.23,A -85,B 0,C 180,E1 -6645,E2 -6645} C_VEL
LIN {X 0,Y 488.808,Z 125.218,A -85,B 0,C 180,E1 -6648.388,E2 -6648.388} C_VEL
LIN {X 0,Y 488.782,Z 125.218,A -85,B 0,C 180,E1 -6651.733,E2 -6651.733} C_VEL
LIN {X 0,Y 488.832,Z 125.219,A -85,B 0,C 180,E1 -6654.224,E2 -6654.224} C_VEL
LIN {X 0,Y 488.955,Z 125.199,A -85,B 0,C 180,E1 -6657.529,E2 -6657.529} C_VEL
LIN {X 0,Y 488.896,Z 125.209,A -85,B 0,C 180,E1 -6660.824,E2 -6660.824} C_VEL
LIN {X 0,Y 488.947,Z 125.207,A -85,B 0,C 180,E1 -6662.472,E2 -6662.472} C_VEL
LIN {X 0,Y 488.829,Z 125.216,A -85,B 0,C 180,E1 -6665.776,E2 -6665.776} C_VEL
LIN {X 0,Y 488.766,Z 125.226,A -85,B 0,C 180,E1 -6668.267,E2 -6668.267} C_VEL
LIN {X 0,Y 488.808,Z 125.221,A -85,B 0,C 180,E1 -6671.612,E2 -6671.612} C_VEL
LIN {X 0,Y 488.751,Z 125.225,A -85,B 0,C 180,E1 -6675.001,E2 -6675.001} C_VEL
LIN {X 0,Y 488.746,Z 125.227,A -85,B 0,C 180,E1 -6678.443,E2 -6678.443} C_VEL
LIN {X 0,Y 488.708,Z 125.229,A -85,B 0,C 180,E1 -6681.071,E2 -6681.071} C_VEL
LIN {X 0,Y 488.672,Z 125.241,A -85,B 0,C 180,E1 -6683.747,E2 -6683.747} C_VEL
LIN {X 0,Y 488.7,Z 125.221,A -85,B 0,C 180,E1 -6686.922,E2 -6686.922} C_VEL
LIN {X 0,Y 488.718,Z 125.23,A -85,B 0,C 180,E1 -6690.22,E2 -6690.22} C_VEL
LIN {X 0,Y 488.711,Z 125.236,A -85,B 0,C 180,E1 -6693.48,E2 -6693.48} C_VEL
LIN {X 0,Y 488.671,Z 125.234,A -85,B 0,C 180,E1 -6696.352,E2 -6696.352} C_VEL
LIN {X 0,Y 488.689,Z 125.238,A -85,B 0,C 180,E1 -6699.256,E2 -6699.256} C_VEL
LIN {X 0,Y 488.667,Z 125.237,A -85,B 0,C 180,E1 -6701.594,E2 -6701.594} C_VEL
LIN {X 0,Y 488.702,Z 125.234,A -85,B 0,C 180,E1 -6704.803,E2 -6704.803} C_VEL
LIN {X 0,Y 488.65,Z 125.242,A -85,B 0,C 180,E1 -6707.47,E2 -6707.47} C_VEL
LIN {X 0,Y 488.704,Z 125.233,A -85,B 0,C 180,E1 -6709.674,E2 -6709.674} C_VEL
LIN {X 0,Y 488.651,Z 125.245,A -85,B 0,C 180,E1 -6712.838,E2 -6712.838} C_VEL
LIN {X 0,Y 488.708,Z 125.233,A -85,B 0,C 180,E1 -6715.885,E2 -6715.885} C_VEL
LIN {X 0,Y 488.658,Z 125.238,A -85,B 0,C 180,E1 -6718.818,E2 -6718.818} C_VEL
LIN {X 0,Y 488.684,Z 125.238,A -85,B 0,C 180,E1 -6721.667,E2 -6721.667} C_VEL
LIN {X 0,Y 488.684,Z 125.241,A -85,B 0,C 180,E1 -6723.074,E2 -6723.074} C_VEL
LIN {X 0,Y 488.511,Z 125.789,A -85,B 0,C 180,E1 -6723.527,E2 -6723.527} C_VEL
LIN {X 0,Y 488.044,Z 127.175,A -85,B 0,C 180,E1 -6723.955,E2 -6723.955} C_VEL
LIN {X 0,Y 486.662,Z 131.367,A -85,B 0,C 180,E1 -6724.744,E2 -6724.744} C_VEL
LIN {X 0,Y 484.922,Z 138.67,A -85,B 0,C 180,E1 -6725.873,E2 -6725.873} C_VEL
LIN {X 0,Y 484.866,Z 140.994,A -85,B 0,C 180,E1 -6726.26,E2 -6726.26} C_VEL
LIN {X 0,Y 484.945,Z 143.632,A -85,B 0,C 180,E1 -6726.658,E2 -6726.658} C_VEL
LIN {X 0,Y 489.109,Z 161.383,A -85,B 0,C 180,E1 -6727.149,E2 -6727.149} C_VEL
LIN {X 0,Y 487.941,Z 275.434,A -85,B 0,C 180,E1 -6728.867,E2 -6728.867} C_VEL
LIN {X 0,Y 487.56,Z 309.699,A -85,B 0,C 180,E1 -6729.413,E2 -6729.413} C_VEL
LIN {X 0,Y 487.181,Z 325.079,A -85,B 0,C 180,E1 -6729.83,E2 -6729.83} C_VEL
LIN {X 0,Y 486.735,Z 339.702,A -85,B 0,C 180,E1 -6730.398,E2 -6730.398} C_VEL
LIN {X 0,Y 486.139,Z 352.112,A -85,B 0,C 180,E1 -6731.018,E2 -6731.018} C_VEL
LIN {X 0,Y 485.411,Z 365.71,A -85,B 0,C 180,E1 -6731.863,E2 -6731.863} C_VEL
LIN {X 0,Y 484.711,Z 378.207,A -85,B 0,C 180,E1 -6732.817,E2 -6732.817} C_VEL
LIN {X 0,Y 484.011,Z 389.462,A -85,B 0,C 180,E1 -6733.843,E2 -6733.843} C_VEL
LIN {X 0,Y 483.312,Z 400.555,A -85,B 0,C 180,E1 -6735.042,E2 -6735.042} C_VEL
LIN {X 0,Y 482.709,Z 410.497,A -85,B 0,C 180,E1 -6736.314,E2 -6736.314} C_VEL
LIN {X 0,Y 482.083,Z 420.118,A -85,B 0,C 180,E1 -6737.781,E2 -6737.781} C_VEL
LIN {X 0,Y 481.693,Z 428.293,A -85,B 0,C 180,E1 -6739.279,E2 -6739.279} C_VEL
LIN {X 0,Y 481.395,Z 434.963,A -85,B 0,C 180,E1 -6740.759,E2 -6740.759} C_VEL
LIN {X 0,Y 481.136,Z 441.143,A -85,B 0,C 180,E1 -6742.446,E2 -6742.446} C_VEL
LIN {X 0,Y 481.045,Z 445.915,A -85,B 0,C 180,E1 -6744.13,E2 -6744.13} C_VEL
LIN {X 0,Y 480.867,Z 449.416,A -85,B 0,C 180,E1 -6745.809,E2 -6745.809} C_VEL
LIN {X 0,Y 480.841,Z 451.732,A -85,B 0,C 180,E1 -6747.487,E2 -6747.487} C_VEL
LIN {X 0,Y 480.757,Z 452.919,A -85,B 0,C 180,E1 -6749.162,E2 -6749.162} C_VEL
LIN {X 0,Y 480.758,Z 452.937,A -85,B 0,C 180,E1 -6750.838,E2 -6750.838} C_VEL
LIN {X 0,Y 480.842,Z 451.821,A -85,B 0,C 180,E1 -6752.513,E2 -6752.513} C_VEL
LIN {X 0,Y 480.867,Z 449.576,A -85,B 0,C 180,E1 -6754.191,E2 -6754.191} C_VEL
LIN {X 0,Y 481.022,Z 446.141,A -85,B 0,C 180,E1 -6755.87,E2 -6755.87} C_VEL
LIN {X 0,Y 481.135,Z 441.441,A -85,B 0,C 180,E1 -6757.554,E2 -6757.554} C_VEL
LIN {X 0,Y 481.374,Z 435.35,A -85,B 0,C 180,E1 -6759.242,E2 -6759.242} C_VEL
LIN {X 0,Y 481.787,Z 427.677,A -85,B 0,C 180,E1 -6760.932,E2 -6760.932} C_VEL
LIN {X 0,Y 482.194,Z 419.355,A -85,B 0,C 180,E1 -6762.438,E2 -6762.438} C_VEL
LIN {X 0,Y 482.753,Z 409.639,A -85,B 0,C 180,E1 -6763.899,E2 -6763.899} C_VEL
LIN {X 0,Y 483.412,Z 399.528,A -85,B 0,C 180,E1 -6765.17,E2 -6765.17} C_VEL
LIN {X 0,Y 484.131,Z 387.91,A -85,B 0,C 180,E1 -6766.401,E2 -6766.401} C_VEL
LIN {X 0,Y 484.817,Z 375.422,A -85,B 0,C 180,E1 -6767.506,E2 -6767.506} C_VEL
LIN {X 0,Y 485.616,Z 362.303,A -85,B 0,C 180,E1 -6768.456,E2 -6768.456} C_VEL
LIN {X 0,Y 486.246,Z 349.808,A -85,B 0,C 180,E1 -6769.197,E2 -6769.197} C_VEL
LIN {X 0,Y 486.877,Z 335.194,A -85,B 0,C 180,E1 -6769.884,E2 -6769.884} C_VEL
LIN {X 0,Y 487.309,Z 320.391,A -85,B 0,C 180,E1 -6770.405,E2 -6770.405} C_VEL
LIN {X 0,Y 487.661,Z 305.79,A -85,B 0,C 180,E1 -6770.754,E2 -6770.754} C_VEL
LIN {X 0,Y 489.086,Z 161.317,A -85,B 0,C 180,E1 -6772.946,E2 -6772.946} C_VEL
LIN {X 0,Y 484.909,Z 143.282,A -85,B 0,C 180,E1 -6773.448,E2 -6773.448} C_VEL
LIN {X 0,Y 484.581,Z 139.11,A -85,B 0,C 180,E1 -6774.164,E2 -6774.164} C_VEL
LIN {X 0,Y 481.634,Z 126.12,A -85,B 0,C 180,E1 -6776.602,E2 -6776.602} C_VEL
LIN {X 0,Y 481.601,Z 126.123,A -85,B 0,C 180,E1 -6779.747,E2 -6779.747} C_VEL
LIN {X 0,Y 481.634,Z 126.116,A -85,B 0,C 180,E1 -6782.677,E2 -6782.677} C_VEL
LIN {X 0,Y 481.642,Z 126.12,A -85,B 0,C 180,E1 -6785.201,E2 -6785.201} C_VEL
LIN {X 0,Y 481.621,Z 126.117,A -85,B 0,C 180,E1 -6788.002,E2 -6788.002} C_VEL
LIN {X 0,Y 481.605,Z 126.122,A -85,B 0,C 180,E1 -6791.047,E2 -6791.047} C_VEL
LIN {X 0,Y 481.651,Z 126.112,A -85,B 0,C 180,E1 -6794.459,E2 -6794.459} C_VEL
LIN {X 0,Y 481.613,Z 126.115,A -85,B 0,C 180,E1 -6796.856,E2 -6796.856} C_VEL
LIN {X 0,Y 481.656,Z 126.11,A -85,B 0,C 180,E1 -6800.057,E2 -6800.057} C_VEL
LIN {X 0,Y 481.61,Z 126.111,A -85,B 0,C 180,E1 -6803.38,E2 -6803.38} C_VEL
LIN {X 0,Y 481.672,Z 126.112,A -85,B 0,C 180,E1 -6806.327,E2 -6806.327} C_VEL
LIN {X 0,Y 481.613,Z 126.107,A -85,B 0,C 180,E1 -6809.426,E2 -6809.426} C_VEL
LIN {X 0,Y 481.646,Z 126.114,A -85,B 0,C 180,E1 -6812.165,E2 -6812.165} C_VEL
LIN {X 0,Y 481.675,Z 126.108,A -85,B 0,C 180,E1 -6814.967,E2 -6814.967} C_VEL
LIN {X 0,Y 481.638,Z 126.111,A -85,B 0,C 180,E1 -6817.704,E2 -6817.704} C_VEL
LIN {X 0,Y 481.695,Z 126.108,A -85,B 0,C 180,E1 -6820.393,E2 -6820.393} C_VEL
LIN {X 0,Y 481.619,Z 126.113,A -85,B 0,C 180,E1 -6823.031,E2 -6823.031} C_VEL
LIN {X 0,Y 481.681,Z 126.108,A -85,B 0,C 180,E1 -6825.638,E2 -6825.638} C_VEL
LIN {X 0,Y 481.754,Z 126.102,A -85,B 0,C 180,E1 -6828.215,E2 -6828.215} C_VEL
LIN {X 0,Y 481.723,Z 126.101,A -85,B 0,C 180,E1 -6831.611,E2 -6831.611} C_VEL
LIN {X 0,Y 481.778,Z 126.095,A -85,B 0,C 180,E1 -6834.139,E2 -6834.139} C_VEL
LIN {X 0,Y 481.911,Z 126.082,A -85,B 0,C 180,E1 -6837.492,E2 -6837.492} C_VEL
LIN {X 0,Y 481.917,Z 126.077,A -85,B 0,C 180,E1 -6840,E2 -6840} C_VEL
LIN {X 0,Y 481.921,Z 126.076,A -85,B 0,C 180,E1 -6842.507,E2 -6842.507} C_VEL
LIN {X 0,Y 481.791,Z 126.095,A -85,B 0,C 180,E1 -6845.861,E2 -6845.861} C_VEL
LIN {X 0,Y 481.739,Z 126.097,A -85,B 0,C 180,E1 -6848.389,E2 -6848.389} C_VEL
LIN {X 0,Y 481.754,Z 126.1,A -85,B 0,C 180,E1 -6851.785,E2 -6851.785} C_VEL
LIN {X 0,Y 481.741,Z 126.105,A -85,B 0,C 180,E1 -6855.224,E2 -6855.224} C_VEL
LIN {X 0,Y 481.71,Z 126.102,A -85,B 0,C 180,E1 -6858.722,E2 -6858.722} C_VEL
LIN {X 0,Y 481.647,Z 126.112,A -85,B 0,C 180,E1 -6861.395,E2 -6861.395} C_VEL
LIN {X 0,Y 481.65,Z 126.111,A -85,B 0,C 180,E1 -6864.114,E2 -6864.114} C_VEL
LIN {X 0,Y 481.697,Z 126.109,A -85,B 0,C 180,E1 -6867.127,E2 -6867.127} C_VEL
LIN {X 0,Y 481.675,Z 126.107,A -85,B 0,C 180,E1 -6869.741,E2 -6869.741} C_VEL
LIN {X 0,Y 481.672,Z 126.113,A -85,B 0,C 180,E1 -6872.674,E2 -6872.674} C_VEL
LIN {X 0,Y 481.638,Z 126.112,A -85,B 0,C 180,E1 -6875.709,E2 -6875.709} C_VEL
LIN {X 0,Y 481.672,Z 126.11,A -85,B 0,C 180,E1 -6878.859,E2 -6878.859} C_VEL
LIN {X 0,Y 481.654,Z 126.112,A -85,B 0,C 180,E1 -6881.913,E2 -6881.913} C_VEL
LIN {X 0,Y 481.656,Z 126.114,A -85,B 0,C 180,E1 -6884.458,E2 -6884.458} C_VEL
LIN {X 0,Y 481.649,Z 126.112,A -85,B 0,C 180,E1 -6887.839,E2 -6887.839} C_VEL
LIN {X 0,Y 481.682,Z 126.108,A -85,B 0,C 180,E1 -6890.651,E2 -6890.651} C_VEL
LIN {X 0,Y 481.628,Z 126.114,A -85,B 0,C 180,E1 -6893.376,E2 -6893.376} C_VEL
LIN {X 0,Y 481.711,Z 126.109,A -85,B 0,C 180,E1 -6896.33,E2 -6896.33} C_VEL
LIN {X 0,Y 481.651,Z 126.112,A -85,B 0,C 180,E1 -6899.417,E2 -6899.417} C_VEL
LIN {X 0,Y 481.693,Z 126.186,A -85,B 0,C 180,E1 -6900.286,E2 -6900.286} C_VEL
LIN {X 0,Y 485.111,Z 140.273,A -85,B 0,C 180,E1 -6902.614,E2 -6902.614} C_VEL
LIN {X 0,Y 485.773,Z 143.437,A -85,B 0,C 180,E1 -6903.12,E2 -6903.12} C_VEL
LIN {X 0,Y 485.098,Z 159.289,A -85,B 0,C 180,E1 -6905.407,E2 -6905.407} C_VEL
LIN {X 0,Y 484.714,Z 167.439,A -85,B 0,C 180,E1 -6906.573,E2 -6906.573} C_VEL
LIN {X 0,Y 488.97,Z 189.672,A -85,B 0,C 180,E1 -6907.143,E2 -6907.143} C_VEL
LIN {X 0,Y 487.419,Z 334.42,A -85,B 0,C 180,E1 -6909.341,E2 -6909.341} C_VEL
LIN {X 0,Y 486.947,Z 350.189,A -85,B 0,C 180,E1 -6909.756,E2 -6909.756} C_VEL
LIN {X 0,Y 486.406,Z 365.245,A -85,B 0,C 180,E1 -6910.332,E2 -6910.332} C_VEL
LIN {X 0,Y 485.725,Z 378.684,A -85,B 0,C 180,E1 -6911.001,E2 -6911.001} C_VEL
LIN {X 0,Y 484.989,Z 392.196,A -85,B 0,C 180,E1 -6911.847,E2 -6911.847} C_VEL
LIN {X 0,Y 484.246,Z 404.659,A -85,B 0,C 180,E1 -6912.8,E2 -6912.8} C_VEL
LIN {X 0,Y 483.523,Z 417.338,A -85,B 0,C 180,E1 -6913.968,E2 -6913.968} C_VEL
LIN {X 0,Y 482.779,Z 428.857,A -85,B 0,C 180,E1 -6915.241,E2 -6915.241} C_VEL
LIN {X 0,Y 482.245,Z 438.557,A -85,B 0,C 180,E1 -6916.516,E2 -6916.516} C_VEL
LIN {X 0,Y 481.775,Z 447.786,A -85,B 0,C 180,E1 -6917.95,E2 -6917.95} C_VEL
LIN {X 0,Y 481.44,Z 456.027,A -85,B 0,C 180,E1 -6919.486,E2 -6919.486} C_VEL
LIN {X 0,Y 481.096,Z 463.439,A -85,B 0,C 180,E1 -6921.177,E2 -6921.177} C_VEL
LIN {X 0,Y 480.983,Z 469.323,A -85,B 0,C 180,E1 -6922.865,E2 -6922.865} C_VEL
LIN {X 0,Y 480.878,Z 472.818,A -85,B 0,C 180,E1 -6924.128,E2 -6924.128} C_VEL
LIN {X 0,Y 480.774,Z 476.351,A -85,B 0,C 180,E1 -6925.808,E2 -6925.808} C_VEL
LIN {X 0,Y 480.818,Z 478.678,A -85,B 0,C 180,E1 -6927.487,E2 -6927.487} C_VEL
LIN {X 0,Y 480.756,Z 479.847,A -85,B 0,C 180,E1 -6929.162,E2 -6929.162} C_VEL
LIN {X 0,Y 480.756,Z 479.846,A -85,B 0,C 180,E1 -6930.838,E2 -6930.838} C_VEL
LIN {X 0,Y 480.818,Z 478.674,A -85,B 0,C 180,E1 -6932.513,E2 -6932.513} C_VEL
LIN {X 0,Y 480.774,Z 476.347,A -85,B 0,C 180,E1 -6934.191,E2 -6934.191} C_VEL
LIN {X 0,Y 480.884,Z 472.82,A -85,B 0,C 180,E1 -6935.872,E2 -6935.872} C_VEL
LIN {X 0,Y 480.984,Z 467.999,A -85,B 0,C 180,E1 -6937.557,E2 -6937.557} C_VEL
LIN {X 0,Y 481.167,Z 461.755,A -85,B 0,C 180,E1 -6939.246,E2 -6939.246} C_VEL
LIN {X 0,Y 481.544,Z 453.917,A -85,B 0,C 180,E1 -6940.937,E2 -6940.937} C_VEL
LIN {X 0,Y 481.809,Z 446.086,A -85,B 0,C 180,E1 -6942.341,E2 -6942.341} C_VEL
LIN {X 0,Y 482.437,Z 435.538,A -85,B 0,C 180,E1 -6943.908,E2 -6943.908} C_VEL
LIN {X 0,Y 482.974,Z 425.268,A -85,B 0,C 180,E1 -6945.184,E2 -6945.184} C_VEL
LIN {X 0,Y 483.782,Z 412.533,A -85,B 0,C 180,E1 -6946.505,E2 -6946.505} C_VEL
LIN {X 0,Y 484.543,Z 399.429,A -85,B 0,C 180,E1 -6947.625,E2 -6947.625} C_VEL
LIN {X 0,Y 485.355,Z 385.788,A -85,B 0,C 180,E1 -6948.576,E2 -6948.576} C_VEL
LIN {X 0,Y 486.064,Z 371.66,A -85,B 0,C 180,E1 -6949.369,E2 -6949.369} C_VEL
LIN {X 0,Y 486.716,Z 357.053,A -85,B 0,C 180,E1 -6950.004,E2 -6950.004} C_VEL
LIN {X 0,Y 487.223,Z 341.955,A -85,B 0,C 180,E1 -6950.483,E2 -6950.483} C_VEL
LIN {X 0,Y 487.564,Z 327.005,A -85,B 0,C 180,E1 -6950.791,E2 -6950.791} C_VEL
LIN {X 0,Y 488.966,Z 189.897,A -85,B 0,C 180,E1 -6952.852,E2 -6952.852} C_VEL
LIN {X 0,Y 484.693,Z 167.386,A -85,B 0,C 180,E1 -6953.432,E2 -6953.432} C_VEL
LIN {X 0,Y 485.834,Z 144.995,A -85,B 0,C 180,E1 -6956.644,E2 -6956.644} C_VEL
LIN {X 0,Y 484.736,Z 138.665,A -85,B 0,C 180,E1 -6957.643,E2 -6957.643} C_VEL
LIN {X 0,Y 481.693,Z 126.11,A -85,B 0,C 180,E1 -6959.74,E2 -6959.74} C_VEL
LIN {X 0,Y 481.672,Z 126.103,A -85,B 0,C 180,E1 -6962.674,E2 -6962.674} C_VEL
LIN {X 0,Y 481.637,Z 126.116,A -85,B 0,C 180,E1 -6965.71,E2 -6965.71} C_VEL
LIN {X 0,Y 481.672,Z 126.108,A -85,B 0,C 180,E1 -6968.859,E2 -6968.859} C_VEL
LIN {X 0,Y 481.653,Z 126.115,A -85,B 0,C 180,E1 -6971.913,E2 -6971.913} C_VEL
LIN {X 0,Y 481.656,Z 126.108,A -85,B 0,C 180,E1 -6974.458,E2 -6974.458} C_VEL
LIN {X 0,Y 481.649,Z 126.114,A -85,B 0,C 180,E1 -6977.839,E2 -6977.839} C_VEL
LIN {X 0,Y 481.662,Z 126.108,A -85,B 0,C 180,E1 -6980.654,E2 -6980.654} C_VEL
LIN {X 0,Y 481.628,Z 126.118,A -85,B 0,C 180,E1 -6983.376,E2 -6983.376} C_VEL
LIN {X 0,Y 481.678,Z 126.105,A -85,B 0,C 180,E1 -6986.328,E2 -6986.328} C_VEL
LIN {X 0,Y 481.651,Z 126.112,A -85,B 0,C 180,E1 -6989.418,E2 -6989.418} C_VEL
LIN {X 0,Y 481.691,Z 126.104,A -85,B 0,C 180,E1 -6992.168,E2 -6992.168} C_VEL
LIN {X 0,Y 481.676,Z 126.112,A -85,B 0,C 180,E1 -6994.968,E2 -6994.968} C_VEL
LIN {X 0,Y 481.649,Z 126.111,A -85,B 0,C 180,E1 -6997.705,E2 -6997.705} C_VEL
LIN {X 0,Y 481.704,Z 126.101,A -85,B 0,C 180,E1 -7000.393,E2 -7000.393} C_VEL
LIN {X 0,Y 481.676,Z 126.109,A -85,B 0,C 180,E1 -7003.033,E2 -7003.033} C_VEL
LIN {X 0,Y 481.686,Z 126.106,A -85,B 0,C 180,E1 -7005.639,E2 -7005.639} C_VEL
LIN {X 0,Y 481.754,Z 126.095,A -85,B 0,C 180,E1 -7008.215,E2 -7008.215} C_VEL
LIN {X 0,Y 481.738,Z 126.095,A -85,B 0,C 180,E1 -7011.611,E2 -7011.611} C_VEL
LIN {X 0,Y 481.791,Z 126.095,A -85,B 0,C 180,E1 -7014.139,E2 -7014.139} C_VEL
LIN {X 0,Y 481.922,Z 126.076,A -85,B 0,C 180,E1 -7017.493,E2 -7017.493} C_VEL
LIN {X 0,Y 481.916,Z 126.078,A -85,B 0,C 180,E1 -7020,E2 -7020} C_VEL
LIN {X 0,Y 481.912,Z 126.082,A -85,B 0,C 180,E1 -7022.508,E2 -7022.508} C_VEL
LIN {X 0,Y 481.788,Z 126.094,A -85,B 0,C 180,E1 -7025.861,E2 -7025.861} C_VEL
LIN {X 0,Y 481.724,Z 126.102,A -85,B 0,C 180,E1 -7028.389,E2 -7028.389} C_VEL
LIN {X 0,Y 481.754,Z 126.101,A -85,B 0,C 180,E1 -7031.785,E2 -7031.785} C_VEL
LIN {X 0,Y 481.732,Z 126.1,A -85,B 0,C 180,E1 -7035.225,E2 -7035.225} C_VEL
LIN {X 0,Y 481.707,Z 126.103,A -85,B 0,C 180,E1 -7038.722,E2 -7038.722} C_VEL
LIN {X 0,Y 481.646,Z 126.111,A -85,B 0,C 180,E1 -7041.395,E2 -7041.395} C_VEL
LIN {X 0,Y 481.65,Z 126.11,A -85,B 0,C 180,E1 -7044.115,E2 -7044.115} C_VEL
LIN {X 0,Y 481.654,Z 126.1,A -85,B 0,C 180,E1 -7047.117,E2 -7047.117} C_VEL
LIN {X 0,Y 481.667,Z 126.113,A -85,B 0,C 180,E1 -7049.742,E2 -7049.742} C_VEL
LIN {X 0,Y 481.653,Z 126.11,A -85,B 0,C 180,E1 -7052.676,E2 -7052.676} C_VEL
LIN {X 0,Y 481.629,Z 126.116,A -85,B 0,C 180,E1 -7055.71,E2 -7055.71} C_VEL
LIN {X 0,Y 481.634,Z 126.114,A -85,B 0,C 180,E1 -7058.863,E2 -7058.863} C_VEL
LIN {X 0,Y 481.621,Z 126.112,A -85,B 0,C 180,E1 -7061.908,E2 -7061.908} C_VEL
LIN {X 0,Y 481.655,Z 126.109,A -85,B 0,C 180,E1 -7064.458,E2 -7064.458} C_VEL
LIN {X 0,Y 481.616,Z 126.119,A -85,B 0,C 180,E1 -7066.855,E2 -7066.855} C_VEL
LIN {X 0,Y 481.656,Z 126.111,A -85,B 0,C 180,E1 -7070.057,E2 -7070.057} C_VEL
LIN {X 0,Y 481.609,Z 126.118,A -85,B 0,C 180,E1 -7073.379,E2 -7073.379} C_VEL
LIN {X 0,Y 481.671,Z 126.112,A -85,B 0,C 180,E1 -7076.327,E2 -7076.327} C_VEL
LIN {X 0,Y 481.61,Z 126.109,A -85,B 0,C 180,E1 -7079.426,E2 -7079.426} C_VEL
LIN {X 0,Y 481.642,Z 126.117,A -85,B 0,C 180,E1 -7082.164,E2 -7082.164} C_VEL
LIN {X 0,Y 481.637,Z 126.193,A -85,B 0,C 180,E1 -7083.544,E2 -7083.544} C_VEL
LIN {X 0,Y 484.833,Z 140.498,A -85,B 0,C 180,E1 -7086.176,E2 -7086.176} C_VEL
LIN {X 0,Y 484.866,Z 140.994,A -85,B 0,C 180,E1 -7086.26,E2 -7086.26} C_VEL
LIN {X 0,Y 485.493,Z 143.159,A -85,B 0,C 180,E1 -7086.538,E2 -7086.538} C_VEL
LIN {X 0,Y 487.248,Z 147.156,A -85,B 0,C 180,E1 -7086.815,E2 -7086.815} C_VEL
LIN {X 0,Y 488.188,Z 151.019,A -85,B 0,C 180,E1 -7086.94,E2 -7086.94} C_VEL
LIN {X 0,Y 487.981,Z 153.572,A -85,B 0,C 180,E1 -7086.97,E2 -7086.97} C_VEL
LIN {X 0,Y 483.756,Z 166.18,A -85,B 0,C 180,E1 -7086.951,E2 -7086.951} C_VEL
LIN {X 0,Y 482.515,Z 172.138,A -85,B 0,C 180,E1 -7086.985,E2 -7086.985} C_VEL
LIN {X 0,Y 481.015,Z 308.882,A -85,B 0,C 180,E1 -7089.095,E2 -7089.095} C_VEL
LIN {X 0,Y 480.552,Z 324.694,A -85,B 0,C 180,E1 -7089.517,E2 -7089.517} C_VEL
LIN {X 0,Y 480.062,Z 340.077,A -85,B 0,C 180,E1 -7090.122,E2 -7090.122} C_VEL
LIN {X 0,Y 479.345,Z 354.215,A -85,B 0,C 180,E1 -7090.849,E2 -7090.849} C_VEL
LIN {X 0,Y 478.568,Z 367.478,A -85,B 0,C 180,E1 -7091.705,E2 -7091.705} C_VEL
LIN {X 0,Y 477.755,Z 380.954,A -85,B 0,C 180,E1 -7092.78,E2 -7092.78} C_VEL
LIN {X 0,Y 476.939,Z 393.173,A -85,B 0,C 180,E1 -7093.961,E2 -7093.961} C_VEL
LIN {X 0,Y 476.216,Z 404.297,A -85,B 0,C 180,E1 -7095.252,E2 -7095.252} C_VEL
LIN {X 0,Y 475.481,Z 415.105,A -85,B 0,C 180,E1 -7096.756,E2 -7096.756} C_VEL
LIN {X 0,Y 474.971,Z 424.067,A -85,B 0,C 180,E1 -7098.261,E2 -7098.261} C_VEL
LIN {X 0,Y 474.497,Z 431.497,A -85,B 0,C 180,E1 -7099.762,E2 -7099.762} C_VEL
LIN {X 0,Y 474.209,Z 438.44,A -85,B 0,C 180,E1 -7101.477,E2 -7101.477} C_VEL
LIN {X 0,Y 473.973,Z 443.898,A -85,B 0,C 180,E1 -7103.187,E2 -7103.187} C_VEL
LIN {X 0,Y 473.822,Z 448.02,A -85,B 0,C 180,E1 -7104.894,E2 -7104.894} C_VEL
LIN {X 0,Y 473.814,Z 450.916,A -85,B 0,C 180,E1 -7106.599,E2 -7106.599} C_VEL
LIN {X 0,Y 473.724,Z 452.663,A -85,B 0,C 180,E1 -7108.3,E2 -7108.3} C_VEL
LIN {X 0,Y 473.669,Z 453.275,A -85,B 0,C 180,E1 -7110,E2 -7110} C_VEL
LIN {X 0,Y 473.725,Z 452.716,A -85,B 0,C 180,E1 -7111.7,E2 -7111.7} C_VEL
LIN {X 0,Y 473.815,Z 451.039,A -85,B 0,C 180,E1 -7113.401,E2 -7113.401} C_VEL
LIN {X 0,Y 473.818,Z 448.21,A -85,B 0,C 180,E1 -7115.106,E2 -7115.106} C_VEL
LIN {X 0,Y 473.969,Z 444.155,A -85,B 0,C 180,E1 -7116.813,E2 -7116.813} C_VEL
LIN {X 0,Y 474.202,Z 438.777,A -85,B 0,C 180,E1 -7118.523,E2 -7118.523} C_VEL
LIN {X 0,Y 474.474,Z 431.925,A -85,B 0,C 180,E1 -7120.239,E2 -7120.239} C_VEL
LIN {X 0,Y 474.959,Z 424.55,A -85,B 0,C 180,E1 -7121.739,E2 -7121.739} C_VEL
LIN {X 0,Y 475.433,Z 415.669,A -85,B 0,C 180,E1 -7123.246,E2 -7123.246} C_VEL
LIN {X 0,Y 476.019,Z 406.611,A -85,B 0,C 180,E1 -7124.536,E2 -7124.536} C_VEL
LIN {X 0,Y 476.727,Z 395.923,A -85,B 0,C 180,E1 -7125.827,E2 -7125.827} C_VEL
LIN {X 0,Y 477.527,Z 384.312,A -85,B 0,C 180,E1 -7127.003,E2 -7127.003} C_VEL
LIN {X 0,Y 478.319,Z 371.506,A -85,B 0,C 180,E1 -7128.083,E2 -7128.083} C_VEL
LIN {X 0,Y 479.12,Z 357.438,A -85,B 0,C 180,E1 -7129.049,E2 -7129.049} C_VEL
LIN {X 0,Y 479.837,Z 344.041,A -85,B 0,C 180,E1 -7129.783,E2 -7129.783} C_VEL
LIN {X 0,Y 480.423,Z 329.016,A -85,B 0,C 180,E1 -7130.421,E2 -7130.421} C_VEL
LIN {X 0,Y 480.851,Z 314.979,A -85,B 0,C 180,E1 -7130.855,E2 -7130.855} C_VEL
LIN {X 0,Y 481.128,Z 299.037,A -85,B 0,C 180,E1 -7131.172,E2 -7131.172} C_VEL
LIN {X 0,Y 482.607,Z 163.442,A -85,B 0,C 180,E1 -7133.24,E2 -7133.24} C_VEL
LIN {X 0,Y 478.531,Z 145.243,A -85,B 0,C 180,E1 -7133.744,E2 -7133.744} C_VEL
LIN {X 0,Y 478.084,Z 143.455,A -85,B 0,C 180,E1 -7133.807,E2 -7133.807} C_VEL
LIN {X 0,Y 476.443,Z 135.131,A -85,B 0,C 180,E1 -7135.327,E2 -7135.327} C_VEL
LIN {X 0,Y 474.612,Z 126.995,A -85,B 0,C 180,E1 -7136.907,E2 -7136.907} C_VEL
LIN {X 0,Y 474.55,Z 126.998,A -85,B 0,C 180,E1 -7140.234,E2 -7140.234} C_VEL
LIN {X 0,Y 474.608,Z 126.995,A -85,B 0,C 180,E1 -7143.223,E2 -7143.223} C_VEL
LIN {X 0,Y 474.566,Z 126.994,A -85,B 0,C 180,E1 -7146.326,E2 -7146.326} C_VEL
LIN {X 0,Y 474.598,Z 126.988,A -85,B 0,C 180,E1 -7149.551,E2 -7149.551} C_VEL
LIN {X 0,Y 474.566,Z 126.999,A -85,B 0,C 180,E1 -7152.94,E2 -7152.94} C_VEL
LIN {X 0,Y 474.581,Z 126.991,A -85,B 0,C 180,E1 -7155.892,E2 -7155.892} C_VEL
LIN {X 0,Y 474.6,Z 126.994,A -85,B 0,C 180,E1 -7159.045,E2 -7159.045} C_VEL
LIN {X 0,Y 474.591,Z 126.985,A -85,B 0,C 180,E1 -7161.707,E2 -7161.707} C_VEL
LIN {X 0,Y 474.613,Z 126.992,A -85,B 0,C 180,E1 -7164.725,E2 -7164.725} C_VEL
LIN {X 0,Y 474.623,Z 126.98,A -85,B 0,C 180,E1 -7167.787,E2 -7167.787} C_VEL
LIN {X 0,Y 474.577,Z 126.994,A -85,B 0,C 180,E1 -7170.896,E2 -7170.896} C_VEL
LIN {X 0,Y 474.591,Z 126.988,A -85,B 0,C 180,E1 -7173.624,E2 -7173.624} C_VEL
LIN {X 0,Y 474.636,Z 126.985,A -85,B 0,C 180,E1 -7176.642,E2 -7176.642} C_VEL
LIN {X 0,Y 474.645,Z 126.989,A -85,B 0,C 180,E1 -7180.089,E2 -7180.089} C_VEL
LIN {X 0,Y 474.595,Z 126.989,A -85,B 0,C 180,E1 -7182.772,E2 -7182.772} C_VEL
LIN {X 0,Y 474.639,Z 126.983,A -85,B 0,C 180,E1 -7185.421,E2 -7185.421} C_VEL
LIN {X 0,Y 474.708,Z 126.982,A -85,B 0,C 180,E1 -7188.038,E2 -7188.038} C_VEL
LIN {X 0,Y 474.699,Z 126.974,A -85,B 0,C 180,E1 -7191.486,E2 -7191.486} C_VEL
LIN {X 0,Y 474.741,Z 126.973,A -85,B 0,C 180,E1 -7194.052,E2 -7194.052} C_VEL
LIN {X 0,Y 474.876,Z 126.957,A -85,B 0,C 180,E1 -7197.455,E2 -7197.455} C_VEL
LIN {X 0,Y 474.886,Z 126.953,A -85,B 0,C 180,E1 -7200,E2 -7200} C_VEL
LIN {X 0,Y 474.887,Z 126.952,A -85,B 0,C 180,E1 -7202.545,E2 -7202.545} C_VEL
LIN {X 0,Y 474.752,Z 126.971,A -85,B 0,C 180,E1 -7205.948,E2 -7205.948} C_VEL
LIN {X 0,Y 474.711,Z 126.973,A -85,B 0,C 180,E1 -7208.514,E2 -7208.514} C_VEL
LIN {X 0,Y 474.708,Z 126.976,A -85,B 0,C 180,E1 -7211.962,E2 -7211.962} C_VEL
LIN {X 0,Y 474.682,Z 126.981,A -85,B 0,C 180,E1 -7215.767,E2 -7215.767} C_VEL
LIN {X 0,Y 474.664,Z 126.983,A -85,B 0,C 180,E1 -7219.01,E2 -7219.01} C_VEL
LIN {X 0,Y 474.59,Z 126.988,A -85,B 0,C 180,E1 -7221.729,E2 -7221.729} C_VEL
LIN {X 0,Y 474.629,Z 126.988,A -85,B 0,C 180,E1 -7224.494,E2 -7224.494} C_VEL
LIN {X 0,Y 474.639,Z 126.986,A -85,B 0,C 180,E1 -7227.324,E2 -7227.324} C_VEL
LIN {X 0,Y 474.604,Z 126.99,A -85,B 0,C 180,E1 -7230.23,E2 -7230.23} C_VEL
LIN {X 0,Y 474.627,Z 126.983,A -85,B 0,C 180,E1 -7233.221,E2 -7233.221} C_VEL
LIN {X 0,Y 474.59,Z 126.994,A -85,B 0,C 180,E1 -7236.323,E2 -7236.323} C_VEL
LIN {X 0,Y 474.619,Z 126.985,A -85,B 0,C 180,E1 -7239.646,E2 -7239.646} C_VEL
LIN {X 0,Y 474.616,Z 126.989,A -85,B 0,C 180,E1 -7242.934,E2 -7242.934} C_VEL
LIN {X 0,Y 474.608,Z 126.99,A -85,B 0,C 180,E1 -7245.895,E2 -7245.895} C_VEL
LIN {X 0,Y 474.629,Z 126.981,A -85,B 0,C 180,E1 -7249.041,E2 -7249.041} C_VEL
LIN {X 0,Y 474.611,Z 126.989,A -85,B 0,C 180,E1 -7251.704,E2 -7251.704} C_VEL
LIN {X 0,Y 474.625,Z 126.988,A -85,B 0,C 180,E1 -7254.725,E2 -7254.725} C_VEL
LIN {X 0,Y 474.636,Z 126.99,A -85,B 0,C 180,E1 -7257.788,E2 -7257.788} C_VEL
LIN {X 0,Y 474.623,Z 127.006,A -85,B 0,C 180,E1 -7259.955,E2 -7259.955} C_VEL
LIN {X 0,Y 478.233,Z 141.814,A -85,B 0,C 180,E1 -7262.448,E2 -7262.448} C_VEL
LIN {X 0,Y 478.988,Z 146.197,A -85,B 0,C 180,E1 -7263.151,E2 -7263.151} C_VEL
LIN {X 0,Y 478.051,Z 164.645,A -85,B 0,C 180,E1 -7265.843,E2 -7265.843} C_VEL
LIN {X 0,Y 477.962,Z 167.606,A -85,B 0,C 180,E1 -7266.236,E2 -7266.236} C_VEL
LIN {X 0,Y 482.401,Z 190.938,A -85,B 0,C 180,E1 -7266.836,E2 -7266.836} C_VEL
LIN {X 0,Y 480.797,Z 334.232,A -85,B 0,C 180,E1 -7269.043,E2 -7269.043} C_VEL
LIN {X 0,Y 480.24,Z 350.273,A -85,B 0,C 180,E1 -7269.471,E2 -7269.471} C_VEL
LIN {X 0,Y 479.689,Z 365.333,A -85,B 0,C 180,E1 -7270.059,E2 -7270.059} C_VEL
LIN {X 0,Y 478.987,Z 378.489,A -85,B 0,C 180,E1 -7270.723,E2 -7270.723} C_VEL
LIN {X 0,Y 478.192,Z 391.999,A -85,B 0,C 180,E1 -7271.58,E2 -7271.58} C_VEL
LIN {X 0,Y 477.326,Z 405.757,A -85,B 0,C 180,E1 -7272.653,E2 -7272.653} C_VEL
LIN {X 0,Y 476.568,Z 418.213,A -85,B 0,C 180,E1 -7273.838,E2 -7273.838} C_VEL
LIN {X 0,Y 475.723,Z 430.429,A -85,B 0,C 180,E1 -7275.236,E2 -7275.236} C_VEL
LIN {X 0,Y 475.055,Z 441.294,A -85,B 0,C 180,E1 -7276.744,E2 -7276.744} C_VEL
LIN {X 0,Y 474.614,Z 450.347,A -85,B 0,C 180,E1 -7278.252,E2 -7278.252} C_VEL
LIN {X 0,Y 474.243,Z 457.856,A -85,B 0,C 180,E1 -7279.756,E2 -7279.756} C_VEL
LIN {X 0,Y 473.977,Z 464.864,A -85,B 0,C 180,E1 -7281.473,E2 -7281.473} C_VEL
LIN {X 0,Y 473.887,Z 470.376,A -85,B 0,C 180,E1 -7283.186,E2 -7283.186} C_VEL
LIN {X 0,Y 473.778,Z 474.543,A -85,B 0,C 180,E1 -7284.894,E2 -7284.894} C_VEL
LIN {X 0,Y 473.739,Z 477.464,A -85,B 0,C 180,E1 -7286.598,E2 -7286.598} C_VEL
LIN {X 0,Y 473.695,Z 479.206,A -85,B 0,C 180,E1 -7288.3,E2 -7288.3} C_VEL
LIN {X 0,Y 473.667,Z 479.803,A -85,B 0,C 180,E1 -7290,E2 -7290} C_VEL
LIN {X 0,Y 473.695,Z 479.203,A -85,B 0,C 180,E1 -7291.7,E2 -7291.7} C_VEL
LIN {X 0,Y 473.739,Z 477.459,A -85,B 0,C 180,E1 -7293.402,E2 -7293.402} C_VEL
LIN {X 0,Y 473.779,Z 474.54,A -85,B 0,C 180,E1 -7295.106,E2 -7295.106} C_VEL
LIN {X 0,Y 473.887,Z 470.379,A -85,B 0,C 180,E1 -7296.814,E2 -7296.814} C_VEL
LIN {X 0,Y 473.977,Z 464.863,A -85,B 0,C 180,E1 -7298.527,E2 -7298.527} C_VEL
LIN {X 0,Y 474.243,Z 457.847,A -85,B 0,C 180,E1 -7300.244,E2 -7300.244} C_VEL
LIN {X 0,Y 474.615,Z 450.34,A -85,B 0,C 180,E1 -7301.748,E2 -7301.748} C_VEL
LIN {X 0,Y 475.055,Z 441.29,A -85,B 0,C 180,E1 -7303.256,E2 -7303.256} C_VEL
LIN {X 0,Y 475.723,Z 430.421,A -85,B 0,C 180,E1 -7304.764,E2 -7304.764} C_VEL
LIN {X 0,Y 476.535,Z 418.207,A -85,B 0,C 180,E1 -7306.163,E2 -7306.163} C_VEL
LIN {X 0,Y 477.316,Z 405.751,A -85,B 0,C 180,E1 -7307.347,E2 -7307.347} C_VEL
LIN {X 0,Y 478.186,Z 391.975,A -85,B 0,C 180,E1 -7308.421,E2 -7308.421} C_VEL
LIN {X 0,Y 478.994,Z 378.453,A -85,B 0,C 180,E1 -7309.277,E2 -7309.277} C_VEL
LIN {X 0,Y 479.695,Z 365.091,A -85,B 0,C 180,E1 -7309.951,E2 -7309.951} C_VEL
LIN {X 0,Y 480.288,Z 350.207,A -85,B 0,C 180,E1 -7310.528,E2 -7310.528} C_VEL
LIN {X 0,Y 480.745,Z 335.303,A -85,B 0,C 180,E1 -7310.932,E2 -7310.932} C_VEL
LIN {X 0,Y 481.2,Z 301.823,A -85,B 0,C 180,E1 -7311.472,E2 -7311.472} C_VEL
LIN {X 0,Y 482.418,Z 190.793,A -85,B 0,C 180,E1 -7313.163,E2 -7313.163} C_VEL
LIN {X 0,Y 477.908,Z 167.188,A -85,B 0,C 180,E1 -7313.785,E2 -7313.785} C_VEL
LIN {X 0,Y 478.979,Z 147.297,A -85,B 0,C 180,E1 -7316.681,E2 -7316.681} C_VEL
LIN {X 0,Y 478.558,Z 143.297,A -85,B 0,C 180,E1 -7317.306,E2 -7317.306} C_VEL
LIN {X 0,Y 475.1,Z 128.955,A -85,B 0,C 180,E1 -7319.706,E2 -7319.706} C_VEL
LIN {X 0,Y 474.635,Z 126.989,A -85,B 0,C 180,E1 -7320.044,E2 -7320.044} C_VEL
LIN {X 0,Y 474.643,Z 126.978,A -85,B 0,C 180,E1 -7323.22,E2 -7323.22} C_VEL
LIN {X 0,Y 474.589,Z 126.994,A -85,B 0,C 180,E1 -7326.324,E2 -7326.324} C_VEL
LIN {X 0,Y 474.628,Z 126.99,A -85,B 0,C 180,E1 -7329.648,E2 -7329.648} C_VEL
LIN {X 0,Y 474.615,Z 126.986,A -85,B 0,C 180,E1 -7332.934,E2 -7332.934} C_VEL
LIN {X 0,Y 474.607,Z 126.991,A -85,B 0,C 180,E1 -7335.895,E2 -7335.895} C_VEL
LIN {X 0,Y 474.628,Z 126.986,A -85,B 0,C 180,E1 -7339.041,E2 -7339.041} C_VEL
LIN {X 0,Y 474.611,Z 126.99,A -85,B 0,C 180,E1 -7341.704,E2 -7341.704} C_VEL
LIN {X 0,Y 474.624,Z 126.983,A -85,B 0,C 180,E1 -7344.726,E2 -7344.726} C_VEL
LIN {X 0,Y 474.636,Z 126.985,A -85,B 0,C 180,E1 -7347.788,E2 -7347.788} C_VEL
LIN {X 0,Y 474.623,Z 126.986,A -85,B 0,C 180,E1 -7350.885,E2 -7350.885} C_VEL
LIN {X 0,Y 474.627,Z 126.987,A -85,B 0,C 180,E1 -7353.626,E2 -7353.626} C_VEL
LIN {X 0,Y 474.636,Z 126.985,A -85,B 0,C 180,E1 -7356.642,E2 -7356.642} C_VEL
LIN {X 0,Y 474.655,Z 126.978,A -85,B 0,C 180,E1 -7360.09,E2 -7360.09} C_VEL
LIN {X 0,Y 474.637,Z 126.989,A -85,B 0,C 180,E1 -7362.774,E2 -7362.774} C_VEL
LIN {X 0,Y 474.646,Z 126.984,A -85,B 0,C 180,E1 -7365.421,E2 -7365.421} C_VEL
LIN {X 0,Y 474.707,Z 126.972,A -85,B 0,C 180,E1 -7368.038,E2 -7368.038} C_VEL
LIN {X 0,Y 474.711,Z 126.97,A -85,B 0,C 180,E1 -7371.486,E2 -7371.486} C_VEL
LIN {X 0,Y 474.743,Z 126.971,A -85,B 0,C 180,E1 -7374.904,E2 -7374.904} C_VEL
LIN {X 0,Y 474.887,Z 126.952,A -85,B 0,C 180,E1 -7377.455,E2 -7377.455} C_VEL
LIN {X 0,Y 474.886,Z 126.954,A -85,B 0,C 180,E1 -7380,E2 -7380} C_VEL
LIN {X 0,Y 474.877,Z 126.958,A -85,B 0,C 180,E1 -7382.545,E2 -7382.545} C_VEL
LIN {X 0,Y 474.749,Z 126.971,A -85,B 0,C 180,E1 -7385.948,E2 -7385.948} C_VEL
LIN {X 0,Y 474.7,Z 126.975,A -85,B 0,C 180,E1 -7388.514,E2 -7388.514} C_VEL
LIN {X 0,Y 474.707,Z 126.981,A -85,B 0,C 180,E1 -7391.962,E2 -7391.962} C_VEL
LIN {X 0,Y 474.691,Z 126.979,A -85,B 0,C 180,E1 -7395.456,E2 -7395.456} C_VEL
LIN {X 0,Y 474.661,Z 126.981,A -85,B 0,C 180,E1 -7399.011,E2 -7399.011} C_VEL
LIN {X 0,Y 474.589,Z 126.993,A -85,B 0,C 180,E1 -7401.729,E2 -7401.729} C_VEL
LIN {X 0,Y 474.628,Z 126.982,A -85,B 0,C 180,E1 -7404.495,E2 -7404.495} C_VEL
LIN {X 0,Y 474.601,Z 126.98,A -85,B 0,C 180,E1 -7407.326,E2 -7407.326} C_VEL
LIN {X 0,Y 474.596,Z 126.989,A -85,B 0,C 180,E1 -7410.231,E2 -7410.231} C_VEL
LIN {X 0,Y 474.616,Z 126.991,A -85,B 0,C 180,E1 -7413.222,E2 -7413.222} C_VEL
LIN {X 0,Y 474.583,Z 126.989,A -85,B 0,C 180,E1 -7416.324,E2 -7416.324} C_VEL
LIN {X 0,Y 474.602,Z 126.989,A -85,B 0,C 180,E1 -7419.644,E2 -7419.644} C_VEL
LIN {X 0,Y 474.57,Z 126.994,A -85,B 0,C 180,E1 -7422.939,E2 -7422.939} C_VEL
LIN {X 0,Y 474.602,Z 126.988,A -85,B 0,C 180,E1 -7425.894,E2 -7425.894} C_VEL
LIN {X 0,Y 474.591,Z 126.995,A -85,B 0,C 180,E1 -7429.339,E2 -7429.339} C_VEL
LIN {X 0,Y 474.59,Z 126.989,A -85,B 0,C 180,E1 -7431.707,E2 -7431.707} C_VEL
LIN {X 0,Y 474.61,Z 126.989,A -85,B 0,C 180,E1 -7434.724,E2 -7434.724} C_VEL
LIN {X 0,Y 474.61,Z 126.989,A -85,B 0,C 180,E1 -7437.786,E2 -7437.786} C_VEL
LIN {X 0,Y 474.575,Z 126.987,A -85,B 0,C 180,E1 -7440.896,E2 -7440.896} C_VEL
LIN {X 0,Y 474.623,Z 127.057,A -85,B 0,C 180,E1 -7443.241,E2 -7443.241} C_VEL
LIN {X 0,Y 477.695,Z 140.758,A -85,B 0,C 180,E1 -7445.806,E2 -7445.806} C_VEL
LIN {X 0,Y 478.127,Z 143.615,A -85,B 0,C 180,E1 -7446.301,E2 -7446.301} C_VEL
LIN {X 0,Y 482.641,Z 163.11,A -85,B 0,C 180,E1 -7446.849,E2 -7446.849} C_VEL
LIN {X 0,Y 482.515,Z 172.138,A -85,B 0,C 180,E1 -7446.985,E2 -7446.985} C_VEL
LIN {X 0,Y 481.86,Z 177.988,A -85,B 0,C 180,E1 -7447.045,E2 -7447.045} C_VEL
LIN {X 0,Y 476.382,Z 197.055,A -85,B 0,C 180,E1 -7447.069,E2 -7447.069} C_VEL
LIN {X 0,Y 475.725,Z 202.904,A -85,B 0,C 180,E1 -7447.129,E2 -7447.129} C_VEL
LIN {X 0,Y 474.399,Z 309.1,A -85,B 0,C 180,E1 -7448.789,E2 -7448.789} C_VEL
LIN {X 0,Y 473.936,Z 324.6,A -85,B 0,C 180,E1 -7449.207,E2 -7449.207} C_VEL
LIN {X 0,Y 473.421,Z 339.452,A -85,B 0,C 180,E1 -7449.789,E2 -7449.789} C_VEL
LIN {X 0,Y 472.634,Z 354.421,A -85,B 0,C 180,E1 -7450.566,E2 -7450.566} C_VEL
LIN {X 0,Y 471.831,Z 367.683,A -85,B 0,C 180,E1 -7451.435,E2 -7451.435} C_VEL
